LIN {X 0,Y 475.139,Z 541.907,A -85,B 0,C 180,E1 -7392.513,E2 -7392.513} C_VEL
LIN {X 0,Y 475.655,Z 532.628,A -85,B 0,C 180,E1 -7393.892,E2 -7393.892} C_VEL
LIN {X 0,Y 476.259,Z 522.288,A -85,B 0,C 180,E1 -7395.184,E2 -7395.184} C_VEL
LIN {X 0,Y 476.842,Z 512.087,A -85,B 0,C 180,E1 -7396.261,E2 -7396.261} C_VEL
LIN {X 0,Y 477.486,Z 500.079,A -85,B 0,C 180,E1 -7397.34,E2 -7397.34} C_VEL
LIN {X 0,Y 478.192,Z 487.079,A -85,B 0,C 180,E1 -7398.309,E2 -7398.309} C_VEL
LIN {X 0,Y 478.818,Z 472.829,A -85,B 0,C 180,E1 -7399.172,E2 -7399.172} C_VEL
LIN {X 0,Y 479.382,Z 458.904,A -85,B 0,C 180,E1 -7399.836,E2 -7399.836} C_VEL
LIN {X 0,Y 479.815,Z 443.461,A -85,B 0,C 180,E1 -7400.392,E2 -7400.392} C_VEL
LIN {X 0,Y 480.139,Z 428.432,A -85,B 0,C 180,E1 -7400.762,E2 -7400.762} C_VEL
LIN {X 0,Y 482.379,Z 286.852,A -85,B 0,C 180,E1 -7403.143,E2 -7403.143} C_VEL
LIN {X 0,Y 481.637,Z 283.318,A -85,B 0,C 180,E1 -7403.243,E2 -7403.243} C_VEL
LIN {X 0,Y 475.324,Z 267.213,A -85,B 0,C 180,E1 -7403.872,E2 -7403.872} C_VEL
LIN {X 0,Y 474.641,Z 263.989,A -85,B 0,C 180,E1 -7404.493,E2 -7404.493} C_VEL
LIN {X 0,Y 474.638,Z 263.985,A -85,B 0,C 180,E1 -7407.323,E2 -7407.323} C_VEL
LIN {X 0,Y 474.602,Z 263.992,A -85,B 0,C 180,E1 -7410.229,E2 -7410.229} C_VEL
LIN {X 0,Y 474.643,Z 263.982,A -85,B 0,C 180,E1 -7413.219,E2 -7413.219} C_VEL
LIN {X 0,Y 474.583,Z 263.992,A -85,B 0,C 180,E1 -7416.323,E2 -7416.323} C_VEL
LIN {X 0,Y 474.624,Z 263.988,A -85,B 0,C 180,E1 -7419.547,E2 -7419.547} C_VEL
LIN {X 0,Y 474.599,Z 263.99,A -85,B 0,C 180,E1 -7422.232,E2 -7422.232} C_VEL
LIN {X 0,Y 474.615,Z 263.987,A -85,B 0,C 180,E1 -7425.296,E2 -7425.296} C_VEL
LIN {X 0,Y 474.616,Z 263.989,A -85,B 0,C 180,E1 -7428.075,E2 -7428.075} C_VEL
LIN {X 0,Y 473.952,Z 264.07,A -85,B 0,C 180,E1 -7428.783,E2 -7428.783} C_VEL
LIN {X 0,Y 471.081,Z 264.432,A -85,B 0,C 180,E1 -7429.933,E2 -7429.933} C_VEL
LIN {X 0,Y 468.659,Z 264.731,A -85,B 0,C 180,E1 -7430.86,E2 -7430.86} C_VEL
LIN {X 0,Y 467.632,Z 264.86,A -85,B 0,C 180,E1 -7431.576,E2 -7431.576} C_VEL
LIN {X 0,Y 467.557,Z 264.869,A -85,B 0,C 180,E1 -7431.819,E2 -7431.819} C_VEL
LIN {X 0,Y 467.554,Z 264.866,A -85,B 0,C 180,E1 -7435.166,E2 -7435.166} C_VEL
LIN {X 0,Y 467.578,Z 264.864,A -85,B 0,C 180,E1 -7438.259,E2 -7438.259} C_VEL
LIN {X 0,Y 467.551,Z 264.867,A -85,B 0,C 180,E1 -7441.248,E2 -7441.248} C_VEL
LIN {X 0,Y 467.58,Z 264.864,A -85,B 0,C 180,E1 -7444.157,E2 -7444.157} C_VEL
LIN {X 0,Y 467.571,Z 264.863,A -85,B 0,C 180,E1 -7446.995,E2 -7446.995} C_VEL
LIN {X 0,Y 467.617,Z 264.864,A -85,B 0,C 180,E1 -7449.776,E2 -7449.776} C_VEL
LIN {X 0,Y 467.592,Z 264.86,A -85,B 0,C 180,E1 -7452.505,E2 -7452.505} C_VEL
LIN {X 0,Y 467.599,Z 264.862,A -85,B 0,C 180,E1 -7455.195,E2 -7455.195} C_VEL
LIN {X 0,Y 467.649,Z 264.858,A -85,B 0,C 180,E1 -7457.853,E2 -7457.853} C_VEL
LIN {X 0,Y 467.674,Z 264.855,A -85,B 0,C 180,E1 -7461.356,E2 -7461.356} C_VEL
LIN {X 0,Y 467.726,Z 264.847,A -85,B 0,C 180,E1 -7463.961,E2 -7463.961} C_VEL
LIN {X 0,Y 467.849,Z 264.834,A -85,B 0,C 180,E1 -7467.416,E2 -7467.416} C_VEL
LIN {X 0,Y 467.872,Z 264.828,A -85,B 0,C 180,E1 -7469.999,E2 -7469.999} C_VEL
LIN {X 0,Y 467.849,Z 264.828,A -85,B 0,C 180,E1 -7472.582,E2 -7472.582} C_VEL
LIN {X 0,Y 467.724,Z 264.845,A -85,B 0,C 180,E1 -7476.036,E2 -7476.036} C_VEL
LIN {X 0,Y 467.67,Z 264.85,A -85,B 0,C 180,E1 -7478.642,E2 -7478.642} C_VEL
LIN {X 0,Y 467.645,Z 264.854,A -85,B 0,C 180,E1 -7482.144,E2 -7482.144} C_VEL
LIN {X 0,Y 467.628,Z 264.861,A -85,B 0,C 180,E1 -7485.694,E2 -7485.694} C_VEL
LIN {X 0,Y 467.605,Z 264.859,A -85,B 0,C 180,E1 -7488.764,E2 -7488.764} C_VEL
LIN {X 0,Y 467.568,Z 264.869,A -85,B 0,C 180,E1 -7491.267,E2 -7491.267} C_VEL
LIN {X 0,Y 467.55,Z 264.867,A -85,B 0,C 180,E1 -7493.943,E2 -7493.943} C_VEL
LIN {X 0,Y 467.599,Z 264.86,A -85,B 0,C 180,E1 -7496.8,E2 -7496.8} C_VEL
LIN {X 0,Y 467.541,Z 264.87,A -85,B 0,C 180,E1 -7499.737,E2 -7499.737} C_VEL
LIN {X 0,Y 467.57,Z 264.864,A -85,B 0,C 180,E1 -7502.758,E2 -7502.758} C_VEL
LIN {X 0,Y 467.542,Z 264.868,A -85,B 0,C 180,E1 -7505.889,E2 -7505.889} C_VEL
LIN {X 0,Y 467.568,Z 264.869,A -85,B 0,C 180,E1 -7509.144,E2 -7509.144} C_VEL
LIN {X 0,Y 467.572,Z 264.863,A -85,B 0,C 180,E1 -7512.566,E2 -7512.566} C_VEL
LIN {X 0,Y 467.556,Z 264.87,A -85,B 0,C 180,E1 -7515.053,E2 -7515.053} C_VEL
LIN {X 0,Y 467.575,Z 264.868,A -85,B 0,C 180,E1 -7517.44,E2 -7517.44} C_VEL
LIN {X 0,Y 467.567,Z 264.866,A -85,B 0,C 180,E1 -7520.855,E2 -7520.855} C_VEL
LIN {X 0,Y 467.547,Z 264.865,A -85,B 0,C 180,E1 -7524.26,E2 -7524.26} C_VEL
LIN {X 0,Y 467.567,Z 264.87,A -85,B 0,C 180,E1 -7527.321,E2 -7527.321} C_VEL
LIN {X 0,Y 467.555,Z 264.866,A -85,B 0,C 180,E1 -7530.667,E2 -7530.667} C_VEL
LIN {X 0,Y 467.602,Z 264.867,A -85,B 0,C 180,E1 -7533.2,E2 -7533.2} C_VEL
LIN {X 0,Y 467.577,Z 264.863,A -85,B 0,C 180,E1 -7536.468,E2 -7536.468} C_VEL
LIN {X 0,Y 467.609,Z 264.859,A -85,B 0,C 180,E1 -7539.777,E2 -7539.777} C_VEL
LIN {X 0,Y 467.594,Z 264.861,A -85,B 0,C 180,E1 -7542.507,E2 -7542.507} C_VEL
LIN {X 0,Y 467.592,Z 264.867,A -85,B 0,C 180,E1 -7545.197,E2 -7545.197} C_VEL
LIN {X 0,Y 467.641,Z 264.854,A -85,B 0,C 180,E1 -7547.855,E2 -7547.855} C_VEL
LIN {X 0,Y 467.666,Z 264.855,A -85,B 0,C 180,E1 -7551.358,E2 -7551.358} C_VEL
LIN {X 0,Y 467.721,Z 264.844,A -85,B 0,C 180,E1 -7553.963,E2 -7553.963} C_VEL
LIN {X 0,Y 467.845,Z 264.832,A -85,B 0,C 180,E1 -7557.418,E2 -7557.418} C_VEL
LIN {X 0,Y 467.867,Z 264.826,A -85,B 0,C 180,E1 -7560.001,E2 -7560.001} C_VEL
LIN {X 0,Y 467.845,Z 264.831,A -85,B 0,C 180,E1 -7562.584,E2 -7562.584} C_VEL
LIN {X 0,Y 467.721,Z 264.844,A -85,B 0,C 180,E1 -7566.038,E2 -7566.038} C_VEL
LIN {X 0,Y 467.669,Z 264.854,A -85,B 0,C 180,E1 -7568.644,E2 -7568.644} C_VEL
LIN {X 0,Y 467.644,Z 264.854,A -85,B 0,C 180,E1 -7572.146,E2 -7572.146} C_VEL
LIN {X 0,Y 467.627,Z 264.856,A -85,B 0,C 180,E1 -7575.696,E2 -7575.696} C_VEL
LIN {X 0,Y 467.606,Z 264.865,A -85,B 0,C 180,E1 -7578.766,E2 -7578.766} C_VEL
LIN {X 0,Y 467.569,Z 264.866,A -85,B 0,C 180,E1 -7581.269,E2 -7581.269} C_VEL
LIN {X 0,Y 467.56,Z 264.864,A -85,B 0,C 180,E1 -7583.944,E2 -7583.944} C_VEL
LIN {X 0,Y 467.605,Z 264.866,A -85,B 0,C 180,E1 -7586.801,E2 -7586.801} C_VEL
LIN {X 0,Y 467.544,Z 264.866,A -85,B 0,C 180,E1 -7589.739,E2 -7589.739} C_VEL
LIN {X 0,Y 467.574,Z 264.87,A -85,B 0,C 180,E1 -7592.76,E2 -7592.76} C_VEL
LIN {X 0,Y 467.544,Z 264.866,A -85,B 0,C 180,E1 -7595.891,E2 -7595.891} C_VEL
LIN {X 0,Y 467.567,Z 264.867,A -85,B 0,C 180,E1 -7599.147,E2 -7599.147} C_VEL
LIN {X 0,Y 467.579,Z 264.867,A -85,B 0,C 180,E1 -7602.568,E2 -7602.568} C_VEL
LIN {X 0,Y 467.558,Z 264.868,A -85,B 0,C 180,E1 -7605.054,E2 -7605.054} C_VEL
LIN {X 0,Y 467.582,Z 264.862,A -85,B 0,C 180,E1 -7607.441,E2 -7607.441} C_VEL
LIN {X 0,Y 467.575,Z 264.869,A -85,B 0,C 180,E1 -7610.857,E2 -7610.857} C_VEL
LIN {X 0,Y 467.552,Z 264.868,A -85,B 0,C 180,E1 -7614.263,E2 -7614.263} C_VEL
LIN {X 0,Y 467.577,Z 264.864,A -85,B 0,C 180,E1 -7617.322,E2 -7617.322} C_VEL
LIN {X 0,Y 467.622,Z 265.064,A -85,B 0,C 180,E1 -7618.201,E2 -7618.201} C_VEL
LIN {X 0,Y 472.061,Z 282.686,A -85,B 0,C 180,E1 -7621.036,E2 -7621.036} C_VEL
LIN {X 0,Y 472.862,Z 286.344,A -85,B 0,C 180,E1 -7621.603,E2 -7621.603} C_VEL
LIN {X 0,Y 472.082,Z 301.582,A -85,B 0,C 180,E1 -7623.713,E2 -7623.713} C_VEL
LIN {X 0,Y 471.187,Z 317.709,A -85,B 0,C 180,E1 -7625.916,E2 -7625.916} C_VEL
LIN {X 0,Y 475.515,Z 342.088,A -85,B 0,C 180,E1 -7626.586,E2 -7626.586} C_VEL
LIN {X 0,Y 473.469,Z 470.629,A -85,B 0,C 180,E1 -7628.79,E2 -7628.79} C_VEL
LIN {X 0,Y 473.069,Z 489.021,A -85,B 0,C 180,E1 -7629.152,E2 -7629.152} C_VEL
LIN {X 0,Y 472.511,Z 504.975,A -85,B 0,C 180,E1 -7629.646,E2 -7629.646} C_VEL
LIN {X 0,Y 471.834,Z 520.281,A -85,B 0,C 180,E1 -7630.307,E2 -7630.307} C_VEL
LIN {X 0,Y 471.125,Z 533.944,A -85,B 0,C 180,E1 -7631.069,E2 -7631.069} C_VEL
LIN {X 0,Y 470.314,Z 548.109,A -85,B 0,C 180,E1 -7632.05,E2 -7632.05} C_VEL
LIN {X 0,Y 469.588,Z 561.022,A -85,B 0,C 180,E1 -7633.146,E2 -7633.146} C_VEL
LIN {X 0,Y 468.886,Z 572.867,A -85,B 0,C 180,E1 -7634.349,E2 -7634.349} C_VEL
LIN {X 0,Y 468.262,Z 583.736,A -85,B 0,C 180,E1 -7635.663,E2 -7635.663} C_VEL
LIN {X 0,Y 467.737,Z 592.926,A -85,B 0,C 180,E1 -7636.976,E2 -7636.976} C_VEL
LIN {X 0,Y 467.384,Z 601.953,A -85,B 0,C 180,E1 -7638.509,E2 -7638.509} C_VEL
LIN {X 0,Y 467.048,Z 609.45,A -85,B 0,C 180,E1 -7640.036,E2 -7640.036} C_VEL
LIN {X 0,Y 466.857,Z 616.377,A -85,B 0,C 180,E1 -7641.779,E2 -7641.779} C_VEL
LIN {X 0,Y 466.796,Z 620.542,A -85,B 0,C 180,E1 -7643.083,E2 -7643.083} C_VEL
LIN {X 0,Y 466.715,Z 624.893,A -85,B 0,C 180,E1 -7644.817,E2 -7644.817} C_VEL
LIN {X 0,Y 466.715,Z 627.937,A -85,B 0,C 180,E1 -7646.548,E2 -7646.548} C_VEL
LIN {X 0,Y 466.691,Z 629.731,A -85,B 0,C 180,E1 -7648.275,E2 -7648.275} C_VEL
LIN {X 0,Y 466.599,Z 630.303,A -85,B 0,C 180,E1 -7650.001,E2 -7650.001} C_VEL
LIN {X 0,Y 466.693,Z 629.626,A -85,B 0,C 180,E1 -7651.727,E2 -7651.727} C_VEL
LIN {X 0,Y 466.735,Z 627.727,A -85,B 0,C 180,E1 -7653.454,E2 -7653.454} C_VEL
LIN {X 0,Y 466.737,Z 624.572,A -85,B 0,C 180,E1 -7655.185,E2 -7655.185} C_VEL
LIN {X 0,Y 466.749,Z 620.092,A -85,B 0,C 180,E1 -7656.92,E2 -7656.92} C_VEL
LIN {X 0,Y 466.881,Z 614.167,A -85,B 0,C 180,E1 -7658.659,E2 -7658.659} C_VEL
LIN {X 0,Y 467.123,Z 606.626,A -85,B 0,C 180,E1 -7660.402,E2 -7660.402} C_VEL
LIN {X 0,Y 467.36,Z 598.534,A -85,B 0,C 180,E1 -7661.934,E2 -7661.934} C_VEL
LIN {X 0,Y 467.86,Z 588.796,A -85,B 0,C 180,E1 -7663.465,E2 -7663.465} C_VEL
LIN {X 0,Y 468.341,Z 578.857,A -85,B 0,C 180,E1 -7664.781,E2 -7664.781} C_VEL
LIN {X 0,Y 468.959,Z 567.176,A -85,B 0,C 180,E1 -7666.084,E2 -7666.084} C_VEL
LIN {X 0,Y 469.721,Z 554.071,A -85,B 0,C 180,E1 -7667.301,E2 -7667.301} C_VEL
LIN {X 0,Y 470.469,Z 541.328,A -85,B 0,C 180,E1 -7668.284,E2 -7668.284} C_VEL
LIN {X 0,Y 471.174,Z 526.601,A -85,B 0,C 180,E1 -7669.214,E2 -7669.214} C_VEL
LIN {X 0,Y 471.963,Z 511.256,A -85,B 0,C 180,E1 -7669.973,E2 -7669.973} C_VEL
LIN {X 0,Y 472.552,Z 496.207,A -85,B 0,C 180,E1 -7670.539,E2 -7670.539} C_VEL
LIN {X 0,Y 473.101,Z 480.803,A -85,B 0,C 180,E1 -7670.945,E2 -7670.945} C_VEL
LIN {X 0,Y 475.142,Z 376.079,A -85,B 0,C 180,E1 -7672.861,E2 -7672.861} C_VEL
LIN {X 0,Y 475.834,Z 341.657,A -85,B 0,C 180,E1 -7673.539,E2 -7673.539} C_VEL
LIN {X 0,Y 472.404,Z 320.404,A -85,B 0,C 180,E1 -7674.215,E2 -7674.215} C_VEL
LIN {X 0,Y 471.131,Z 313.647,A -85,B 0,C 180,E1 -7674.462,E2 -7674.462} C_VEL
LIN {X 0,Y 472.534,Z 292.625,A -85,B 0,C 180,E1 -7677.457,E2 -7677.457} C_VEL
LIN {X 0,Y 472.897,Z 286.289,A -85,B 0,C 180,E1 -7678.397,E2 -7678.397} C_VEL
LIN {X 0,Y 470.902,Z 276.797,A -85,B 0,C 180,E1 -7680.046,E2 -7680.046} C_VEL
LIN {X 0,Y 467.596,Z 264.869,A -85,B 0,C 180,E1 -7682.355,E2 -7682.355} C_VEL
LIN {X 0,Y 467.569,Z 264.872,A -85,B 0,C 180,E1 -7684.833,E2 -7684.833} C_VEL
LIN {X 0,Y 467.571,Z 264.868,A -85,B 0,C 180,E1 -7688.045,E2 -7688.045} C_VEL
LIN {X 0,Y 467.584,Z 264.868,A -85,B 0,C 180,E1 -7691.277,E2 -7691.277} C_VEL
LIN {X 0,Y 467.56,Z 264.869,A -85,B 0,C 180,E1 -7693.821,E2 -7693.821} C_VEL
LIN {X 0,Y 467.562,Z 264.87,A -85,B 0,C 180,E1 -7696.256,E2 -7696.256} C_VEL
LIN {X 0,Y 467.584,Z 264.867,A -85,B 0,C 180,E1 -7698.723,E2 -7698.723} C_VEL
LIN {X 0,Y 467.568,Z 264.868,A -85,B 0,C 180,E1 -7701.955,E2 -7701.955} C_VEL
LIN {X 0,Y 467.569,Z 264.869,A -85,B 0,C 180,E1 -7705.167,E2 -7705.167} C_VEL
LIN {X 0,Y 467.589,Z 264.868,A -85,B 0,C 180,E1 -7708.26,E2 -7708.26} C_VEL
LIN {X 0,Y 467.562,Z 264.87,A -85,B 0,C 180,E1 -7711.249,E2 -7711.249} C_VEL
LIN {X 0,Y 467.606,Z 264.969,A -85,B 0,C 180,E1 -7713.68,E2 -7713.68} C_VEL
LIN {X 0,Y 469.637,Z 272.657,A -85,B 0,C 180,E1 -7715.539,E2 -7715.539} C_VEL
LIN {X 0,Y 476.247,Z 287.026,A -85,B 0,C 180,E1 -7716.329,E2 -7716.329} C_VEL
LIN {X 0,Y 476.76,Z 288.495,A -85,B 0,C 180,E1 -7716.395,E2 -7716.395} C_VEL
LIN {X 0,Y 474.275,Z 384.716,A -85,B 0,C 180,E1 -7718.256,E2 -7718.256} C_VEL
LIN {X 0,Y 473.345,Z 436.186,A -85,B 0,C 180,E1 -7719.213,E2 -7719.213} C_VEL
LIN {X 0,Y 472.938,Z 451.934,A -85,B 0,C 180,E1 -7719.683,E2 -7719.683} C_VEL
LIN {X 0,Y 472.36,Z 467.317,A -85,B 0,C 180,E1 -7720.328,E2 -7720.328} C_VEL
LIN {X 0,Y 471.792,Z 481.298,A -85,B 0,C 180,E1 -7721.095,E2 -7721.095} C_VEL
LIN {X 0,Y 471.139,Z 494.235,A -85,B 0,C 180,E1 -7721.969,E2 -7721.969} C_VEL
LIN {X 0,Y 470.398,Z 506.614,A -85,B 0,C 180,E1 -7722.98,E2 -7722.98} C_VEL
LIN {X 0,Y 469.693,Z 518.511,A -85,B 0,C 180,E1 -7724.152,E2 -7724.152} C_VEL
LIN {X 0,Y 469.09,Z 529.643,A -85,B 0,C 180,E1 -7725.466,E2 -7725.466} C_VEL
LIN {X 0,Y 468.432,Z 539.004,A -85,B 0,C 180,E1 -7726.773,E2 -7726.773} C_VEL
LIN {X 0,Y 468.011,Z 548.131,A -85,B 0,C 180,E1 -7728.303,E2 -7728.303} C_VEL
LIN {X 0,Y 467.538,Z 555.678,A -85,B 0,C 180,E1 -7729.826,E2 -7729.826} C_VEL
LIN {X 0,Y 467.245,Z 561.874,A -85,B 0,C 180,E1 -7731.349,E2 -7731.349} C_VEL
LIN {X 0,Y 467.029,Z 567.516,A -85,B 0,C 180,E1 -7733.085,E2 -7733.085} C_VEL
LIN {X 0,Y 466.78,Z 571.769,A -85,B 0,C 180,E1 -7734.816,E2 -7734.816} C_VEL
LIN {X 0,Y 466.809,Z 574.726,A -85,B 0,C 180,E1 -7736.547,E2 -7736.547} C_VEL
LIN {X 0,Y 466.698,Z 576.487,A -85,B 0,C 180,E1 -7738.273,E2 -7738.273} C_VEL
LIN {X 0,Y 466.603,Z 577.058,A -85,B 0,C 180,E1 -7739.999,E2 -7739.999} C_VEL
LIN {X 0,Y 466.698,Z 576.411,A -85,B 0,C 180,E1 -7741.725,E2 -7741.725} C_VEL
LIN {X 0,Y 466.798,Z 574.598,A -85,B 0,C 180,E1 -7743.452,E2 -7743.452} C_VEL
LIN {X 0,Y 466.771,Z 571.587,A -85,B 0,C 180,E1 -7745.182,E2 -7745.182} C_VEL
LIN {X 0,Y 466.964,Z 568.154,A -85,B 0,C 180,E1 -7746.618,E2 -7746.618} C_VEL
LIN {X 0,Y 467.113,Z 563.187,A -85,B 0,C 180,E1 -7748.217,E2 -7748.217} C_VEL
LIN {X 0,Y 467.403,Z 556.372,A -85,B 0,C 180,E1 -7749.957,E2 -7749.957} C_VEL
LIN {X 0,Y 467.875,Z 547.853,A -85,B 0,C 180,E1 -7751.699,E2 -7751.699} C_VEL
LIN {X 0,Y 468.343,Z 538.722,A -85,B 0,C 180,E1 -7753.228,E2 -7753.228} C_VEL
LIN {X 0,Y 469.019,Z 527.697,A -85,B 0,C 180,E1 -7754.757,E2 -7754.757} C_VEL
LIN {X 0,Y 469.682,Z 516.311,A -85,B 0,C 180,E1 -7756.07,E2 -7756.07} C_VEL
LIN {X 0,Y 470.414,Z 504.354,A -85,B 0,C 180,E1 -7757.222,E2 -7757.222} C_VEL
LIN {X 0,Y 471.102,Z 491.472,A -85,B 0,C 180,E1 -7758.256,E2 -7758.256} C_VEL
LIN {X 0,Y 471.777,Z 478.174,A -85,B 0,C 180,E1 -7759.13,E2 -7759.13} C_VEL
LIN {X 0,Y 472.413,Z 464.765,A -85,B 0,C 180,E1 -7759.838,E2 -7759.838} C_VEL
LIN {X 0,Y 472.915,Z 449.672,A -85,B 0,C 180,E1 -7760.459,E2 -7760.459} C_VEL
LIN {X 0,Y 473.314,Z 435.541,A -85,B 0,C 180,E1 -7760.876,E2 -7760.876} C_VEL
LIN {X 0,Y 473.668,Z 413.779,A -85,B 0,C 180,E1 -7761.287,E2 -7761.287} C_VEL
LIN {X 0,Y 475.785,Z 287.085,A -85,B 0,C 180,E1 -7763.464,E2 -7763.464} C_VEL
LIN {X 0,Y 468.175,Z 267.585,A -85,B 0,C 180,E1 -7764.228,E2 -7764.228} C_VEL
LIN {X 0,Y 467.608,Z 264.865,A -85,B 0,C 180,E1 -7764.768,E2 -7764.768} C_VEL
LIN {X 0,Y 467.581,Z 264.868,A -85,B 0,C 180,E1 -7767.77,E2 -7767.77} C_VEL
LIN {X 0,Y 467.567,Z 264.865,A -85,B 0,C 180,E1 -7771.043,E2 -7771.043} C_VEL
LIN {X 0,Y 467.588,Z 264.864,A -85,B 0,C 180,E1 -7774.241,E2 -7774.241} C_VEL
LIN {X 0,Y 467.542,Z 264.867,A -85,B 0,C 180,E1 -7777.184,E2 -7777.184} C_VEL
LIN {X 0,Y 467.569,Z 264.866,A -85,B 0,C 180,E1 -7780.264,E2 -7780.264} C_VEL
LIN {X 0,Y 467.547,Z 264.873,A -85,B 0,C 180,E1 -7783.744,E2 -7783.744} C_VEL
LIN {X 0,Y 467.549,Z 264.868,A -85,B 0,C 180,E1 -7786.254,E2 -7786.254} C_VEL
LIN {X 0,Y 467.576,Z 264.862,A -85,B 0,C 180,E1 -7788.722,E2 -7788.722} C_VEL
LIN {X 0,Y 467.557,Z 264.869,A -85,B 0,C 180,E1 -7791.819,E2 -7791.819} C_VEL
LIN {X 0,Y 466.897,Z 264.955,A -85,B 0,C 180,E1 -7792.538,E2 -7792.538} C_VEL
LIN {X 0,Y 464.007,Z 265.314,A -85,B 0,C 180,E1 -7793.705,E2 -7793.705} C_VEL
LIN {X 0,Y 461.585,Z 265.61,A -85,B 0,C 180,E1 -7794.647,E2 -7794.647} C_VEL
LIN {X 0,Y 460.589,Z 265.736,A -85,B 0,C 180,E1 -7795.375,E2 -7795.375} C_VEL
LIN {X 0,Y 460.533,Z 265.746,A -85,B 0,C 180,E1 -7795.621,E2 -7795.621} C_VEL
LIN {X 0,Y 460.533,Z 265.739,A -85,B 0,C 180,E1 -7798.743,E2 -7798.743} C_VEL
LIN {X 0,Y 460.546,Z 265.739,A -85,B 0,C 180,E1 -7802.26,E2 -7802.26} C_VEL
LIN {X 0,Y 460.535,Z 265.739,A -85,B 0,C 180,E1 -7804.703,E2 -7804.703} C_VEL
LIN {X 0,Y 460.505,Z 265.749,A -85,B 0,C 180,E1 -7807.57,E2 -7807.57} C_VEL
LIN {X 0,Y 460.562,Z 265.736,A -85,B 0,C 180,E1 -7810.383,E2 -7810.383} C_VEL
LIN {X 0,Y 460.594,Z 265.735,A -85,B 0,C 180,E1 -7814.001,E2 -7814.001} C_VEL
LIN {X 0,Y 460.602,Z 265.739,A -85,B 0,C 180,E1 -7817.665,E2 -7817.665} C_VEL
LIN {X 0,Y 460.621,Z 265.732,A -85,B 0,C 180,E1 -7821.223,E2 -7821.223} C_VEL
LIN {X 0,Y 460.692,Z 265.724,A -85,B 0,C 180,E1 -7823.869,E2 -7823.869} C_VEL
LIN {X 0,Y 460.79,Z 265.713,A -85,B 0,C 180,E1 -7827.376,E2 -7827.376} C_VEL
LIN {X 0,Y 460.843,Z 265.703,A -85,B 0,C 180,E1 -7829.999,E2 -7829.999} C_VEL
LIN {X 0,Y 460.79,Z 265.707,A -85,B 0,C 180,E1 -7832.621,E2 -7832.621} C_VEL
LIN {X 0,Y 460.691,Z 265.721,A -85,B 0,C 180,E1 -7836.129,E2 -7836.129} C_VEL
LIN {X 0,Y 460.617,Z 265.729,A -85,B 0,C 180,E1 -7838.775,E2 -7838.775} C_VEL
LIN {X 0,Y 460.603,Z 265.731,A -85,B 0,C 180,E1 -7842.444,E2 -7842.444} C_VEL
LIN {X 0,Y 460.589,Z 265.734,A -85,B 0,C 180,E1 -7845.997,E2 -7845.997} C_VEL
LIN {X 0,Y 460.559,Z 265.738,A -85,B 0,C 180,E1 -7848.901,E2 -7848.901} C_VEL
LIN {X 0,Y 460.503,Z 265.751,A -85,B 0,C 180,E1 -7851.485,E2 -7851.485} C_VEL
LIN {X 0,Y 460.518,Z 265.741,A -85,B 0,C 180,E1 -7854.332,E2 -7854.332} C_VEL
LIN {X 0,Y 460.575,Z 265.737,A -85,B 0,C 180,E1 -7857.747,E2 -7857.747} C_VEL
LIN {X 0,Y 460.509,Z 265.749,A -85,B 0,C 180,E1 -7861.283,E2 -7861.283} C_VEL
LIN {X 0,Y 460.52,Z 265.741,A -85,B 0,C 180,E1 -7864.505,E2 -7864.505} C_VEL
LIN {X 0,Y 460.514,Z 265.746,A -85,B 0,C 180,E1 -7867.62,E2 -7867.62} C_VEL
LIN {X 0,Y 460.528,Z 265.74,A -85,B 0,C 180,E1 -7870.269,E2 -7870.269} C_VEL
LIN {X 0,Y 460.495,Z 265.751,A -85,B 0,C 180,E1 -7873.374,E2 -7873.374} C_VEL
LIN {X 0,Y 460.497,Z 265.745,A -85,B 0,C 180,E1 -7876.626,E2 -7876.626} C_VEL
LIN {X 0,Y 460.527,Z 265.742,A -85,B 0,C 180,E1 -7879.73,E2 -7879.73} C_VEL
LIN {X 0,Y 460.485,Z 265.746,A -85,B 0,C 180,E1 -7882.523,E2 -7882.523} C_VEL
LIN {X 0,Y 460.533,Z 265.742,A -85,B 0,C 180,E1 -7885.624,E2 -7885.624} C_VEL
LIN {X 0,Y 460.522,Z 265.743,A -85,B 0,C 180,E1 -7888.745,E2 -7888.745} C_VEL
LIN {X 0,Y 460.566,Z 265.735,A -85,B 0,C 180,E1 -7892.254,E2 -7892.254} C_VEL
LIN {X 0,Y 460.543,Z 265.74,A -85,B 0,C 180,E1 -7894.706,E2 -7894.706} C_VEL
LIN {X 0,Y 460.496,Z 265.747,A -85,B 0,C 180,E1 -7897.572,E2 -7897.572} C_VEL
LIN {X 0,Y 460.555,Z 265.737,A -85,B 0,C 180,E1 -7900.385,E2 -7900.385} C_VEL
LIN {X 0,Y 460.55,Z 265.745,A -85,B 0,C 180,E1 -7903.147,E2 -7903.147} C_VEL
LIN {X 0,Y 460.539,Z 265.739,A -85,B 0,C 180,E1 -7905.868,E2 -7905.868} C_VEL
LIN {X 0,Y 460.596,Z 265.733,A -85,B 0,C 180,E1 -7908.56,E2 -7908.56} C_VEL
LIN {X 0,Y 460.681,Z 265.721,A -85,B 0,C 180,E1 -7912.109,E2 -7912.109} C_VEL
LIN {X 0,Y 460.678,Z 265.725,A -85,B 0,C 180,E1 -7914.749,E2 -7914.749} C_VEL
LIN {X 0,Y 460.81,Z 265.708,A -85,B 0,C 180,E1 -7917.378,E2 -7917.378} C_VEL
LIN {X 0,Y 460.838,Z 265.701,A -85,B 0,C 180,E1 -7920.001,E2 -7920.001} C_VEL
LIN {X 0,Y 460.786,Z 265.711,A -85,B 0,C 180,E1 -7922.623,E2 -7922.623} C_VEL
LIN {X 0,Y 460.688,Z 265.72,A -85,B 0,C 180,E1 -7926.131,E2 -7926.131} C_VEL
LIN {X 0,Y 460.616,Z 265.734,A -85,B 0,C 180,E1 -7928.777,E2 -7928.777} C_VEL
LIN {X 0,Y 460.601,Z 265.733,A -85,B 0,C 180,E1 -7932.446,E2 -7932.446} C_VEL
LIN {X 0,Y 460.588,Z 265.732,A -85,B 0,C 180,E1 -7935.999,E2 -7935.999} C_VEL
LIN {X 0,Y 460.56,Z 265.744,A -85,B 0,C 180,E1 -7938.903,E2 -7938.903} C_VEL
LIN {X 0,Y 460.505,Z 265.744,A -85,B 0,C 180,E1 -7941.487,E2 -7941.487} C_VEL
LIN {X 0,Y 460.527,Z 265.742,A -85,B 0,C 180,E1 -7944.334,E2 -7944.334} C_VEL
LIN {X 0,Y 460.562,Z 265.739,A -85,B 0,C 180,E1 -7947.245,E2 -7947.245} C_VEL
LIN {X 0,Y 460.501,Z 265.745,A -85,B 0,C 180,E1 -7950.241,E2 -7950.241} C_VEL
LIN {X 0,Y 460.519,Z 265.743,A -85,B 0,C 180,E1 -7953.326,E2 -7953.326} C_VEL
LIN {X 0,Y 460.467,Z 265.752,A -85,B 0,C 180,E1 -7956.531,E2 -7956.531} C_VEL
LIN {X 0,Y 460.518,Z 265.741,A -85,B 0,C 180,E1 -7959.864,E2 -7959.864} C_VEL
LIN {X 0,Y 460.505,Z 265.749,A -85,B 0,C 180,E1 -7962.902,E2 -7962.902} C_VEL
LIN {X 0,Y 460.501,Z 265.743,A -85,B 0,C 180,E1 -7965.832,E2 -7965.832} C_VEL
LIN {X 0,Y 460.524,Z 265.747,A -85,B 0,C 180,E1 -7968.99,E2 -7968.99} C_VEL
LIN {X 0,Y 460.519,Z 265.745,A -85,B 0,C 180,E1 -7971.268,E2 -7971.268} C_VEL
LIN {X 0,Y 460.503,Z 265.747,A -85,B 0,C 180,E1 -7974.556,E2 -7974.556} C_VEL
LIN {X 0,Y 460.566,Z 265.837,A -85,B 0,C 180,E1 -7977.863,E2 -7977.863} C_VEL
LIN {X 0,Y 465.166,Z 284.085,A -85,B 0,C 180,E1 -7980.842,E2 -7980.842} C_VEL
LIN {X 0,Y 466.072,Z 289.256,A -85,B 0,C 180,E1 -7981.643,E2 -7981.643} C_VEL
LIN {X 0,Y 464.688,Z 312.945,A -85,B 0,C 180,E1 -7984.947,E2 -7984.947} C_VEL
LIN {X 0,Y 464.42,Z 317.387,A -85,B 0,C 180,E1 -7985.559,E2 -7985.559} C_VEL
LIN {X 0,Y 468.902,Z 342.971,A -85,B 0,C 180,E1 -7986.277,E2 -7986.277} C_VEL
LIN {X 0,Y 466.793,Z 467.854,A -85,B 0,C 180,E1 -7988.472,E2 -7988.472} C_VEL
LIN {X 0,Y 466.329,Z 488.219,A -85,B 0,C 180,E1 -7988.871,E2 -7988.871} C_VEL
LIN {X 0,Y 465.723,Z 504.376,A -85,B 0,C 180,E1 -7989.374,E2 -7989.374} C_VEL
LIN {X 0,Y 465.085,Z 518.991,A -85,B 0,C 180,E1 -7990.009,E2 -7990.009} C_VEL
LIN {X 0,Y 464.304,Z 532.848,A -85,B 0,C 180,E1 -7990.78,E2 -7990.78} C_VEL
LIN {X 0,Y 463.467,Z 547.151,A -85,B 0,C 180,E1 -7991.776,E2 -7991.776} C_VEL
LIN {X 0,Y 462.687,Z 560.161,A -85,B 0,C 180,E1 -7992.886,E2 -7992.886} C_VEL
LIN {X 0,Y 461.949,Z 572.096,A -85,B 0,C 180,E1 -7994.108,E2 -7994.108} C_VEL
LIN {X 0,Y 461.266,Z 583.034,A -85,B 0,C 180,E1 -7995.441,E2 -7995.441} C_VEL
LIN {X 0,Y 460.656,Z 593.691,A -85,B 0,C 180,E1 -7996.997,E2 -7996.997} C_VEL
LIN {X 0,Y 460.276,Z 602.535,A -85,B 0,C 180,E1 -7998.552,E2 -7998.552} C_VEL
LIN {X 0,Y 459.98,Z 608.933,A -85,B 0,C 180,E1 -7999.881,E2 -7999.881} C_VEL
LIN {X 0,Y 459.772,Z 615.901,A -85,B 0,C 180,E1 -8001.652,E2 -8001.652} C_VEL
LIN {X 0,Y 459.715,Z 620.086,A -85,B 0,C 180,E1 -8002.976,E2 -8002.976} C_VEL
LIN {X 0,Y 459.62,Z 624.463,A -85,B 0,C 180,E1 -8004.737,E2 -8004.737} C_VEL
LIN {X 0,Y 459.628,Z 627.523,A -85,B 0,C 180,E1 -8006.495,E2 -8006.495} C_VEL
LIN {X 0,Y 459.627,Z 629.328,A -85,B 0,C 180,E1 -8008.249,E2 -8008.249} C_VEL
LIN {X 0,Y 459.53,Z 629.898,A -85,B 0,C 180,E1 -8010.001,E2 -8010.001} C_VEL
LIN {X 0,Y 459.63,Z 629.216,A -85,B 0,C 180,E1 -8011.754,E2 -8011.754} C_VEL
LIN {X 0,Y 459.646,Z 627.305,A -85,B 0,C 180,E1 -8013.508,E2 -8013.508} C_VEL
LIN {X 0,Y 459.67,Z 624.135,A -85,B 0,C 180,E1 -8015.265,E2 -8015.265} C_VEL
LIN {X 0,Y 459.691,Z 619.625,A -85,B 0,C 180,E1 -8017.026,E2 -8017.026} C_VEL
LIN {X 0,Y 459.8,Z 613.67,A -85,B 0,C 180,E1 -8018.793,E2 -8018.793} C_VEL
LIN {X 0,Y 460.078,Z 606.105,A -85,B 0,C 180,E1 -8020.564,E2 -8020.564} C_VEL
LIN {X 0,Y 460.322,Z 597.852,A -85,B 0,C 180,E1 -8022.14,E2 -8022.14} C_VEL
LIN {X 0,Y 460.85,Z 588.201,A -85,B 0,C 180,E1 -8023.674,E2 -8023.674} C_VEL
LIN {X 0,Y 461.371,Z 578.233,A -85,B 0,C 180,E1 -8025.009,E2 -8025.009} C_VEL
LIN {X 0,Y 462.009,Z 567.012,A -85,B 0,C 180,E1 -8026.282,E2 -8026.282} C_VEL
LIN {X 0,Y 462.762,Z 554.7,A -85,B 0,C 180,E1 -8027.455,E2 -8027.455} C_VEL
LIN {X 0,Y 463.548,Z 542.14,A -85,B 0,C 180,E1 -8028.452,E2 -8028.452} C_VEL
LIN {X 0,Y 464.264,Z 528.702,A -85,B 0,C 180,E1 -8029.339,E2 -8029.339} C_VEL
LIN {X 0,Y 465.063,Z 514.169,A -85,B 0,C 180,E1 -8030.109,E2 -8030.109} C_VEL
LIN {X 0,Y 465.735,Z 499.213,A -85,B 0,C 180,E1 -8030.721,E2 -8030.721} C_VEL
LIN {X 0,Y 466.351,Z 483.738,A -85,B 0,C 180,E1 -8031.177,E2 -8031.177} C_VEL
LIN {X 0,Y 468.815,Z 370.332,A -85,B 0,C 180,E1 -8033.343,E2 -8033.343} C_VEL
LIN {X 0,Y 469.561,Z 343.336,A -85,B 0,C 180,E1 -8033.887,E2 -8033.887} C_VEL
LIN {X 0,Y 466.307,Z 322.533,A -85,B 0,C 180,E1 -8034.572,E2 -8034.572} C_VEL
LIN {X 0,Y 464.456,Z 312.9,A -85,B 0,C 180,E1 -8034.949,E2 -8034.949} C_VEL
LIN {X 0,Y 465.946,Z 292.874,A -85,B 0,C 180,E1 -8037.878,E2 -8037.878} C_VEL
LIN {X 0,Y 466.237,Z 288.569,A -85,B 0,C 180,E1 -8038.529,E2 -8038.529} C_VEL
LIN {X 0,Y 464.501,Z 279.9,A -85,B 0,C 180,E1 -8040.069,E2 -8040.069} C_VEL
LIN {X 0,Y 461.527,Z 269.097,A -85,B 0,C 180,E1 -8042.207,E2 -8042.207} C_VEL
LIN {X 0,Y 460.537,Z 265.749,A -85,B 0,C 180,E1 -8042.931,E2 -8042.931} C_VEL
LIN {X 0,Y 460.503,Z 265.749,A -85,B 0,C 180,E1 -8046.015,E2 -8046.015} C_VEL
LIN {X 0,Y 460.55,Z 265.745,A -85,B 0,C 180,E1 -8048.898,E2 -8048.898} C_VEL
LIN {X 0,Y 460.529,Z 265.745,A -85,B 0,C 180,E1 -8052.182,E2 -8052.182} C_VEL
LIN {X 0,Y 460.523,Z 265.746,A -85,B 0,C 180,E1 -8055.412,E2 -8055.412} C_VEL
LIN {X 0,Y 460.538,Z 265.745,A -85,B 0,C 180,E1 -8058.398,E2 -8058.398} C_VEL
LIN {X 0,Y 460.531,Z 265.745,A -85,B 0,C 180,E1 -8061.267,E2 -8061.267} C_VEL
LIN {X 0,Y 460.515,Z 265.75,A -85,B 0,C 180,E1 -8064.554,E2 -8064.554} C_VEL
LIN {X 0,Y 460.538,Z 265.744,A -85,B 0,C 180,E1 -8067.716,E2 -8067.716} C_VEL
LIN {X 0,Y 460.533,Z 265.747,A -85,B 0,C 180,E1 -8070.768,E2 -8070.768} C_VEL
LIN {X 0,Y 460.541,Z 265.828,A -85,B 0,C 180,E1 -8073.091,E2 -8073.091} C_VEL
LIN {X 0,Y 462.697,Z 273.702,A -85,B 0,C 180,E1 -8075.043,E2 -8075.043} C_VEL
LIN {X 0,Y 469.138,Z 287.071,A -85,B 0,C 180,E1 -8075.848,E2 -8075.848} C_VEL
LIN {X 0,Y 470.442,Z 290.142,A -85,B 0,C 180,E1 -8076.009,E2 -8076.009} C_VEL
LIN {X 0,Y 467.799,Z 384.926,A -85,B 0,C 180,E1 -8077.91,E2 -8077.91} C_VEL
LIN {X 0,Y 466.754,Z 437.046,A -85,B 0,C 180,E1 -8078.912,E2 -8078.912} C_VEL
LIN {X 0,Y 466.287,Z 452.529,A -85,B 0,C 180,E1 -8079.385,E2 -8079.385} C_VEL
LIN {X 0,Y 465.689,Z 467.723,A -85,B 0,C 180,E1 -8080.034,E2 -8080.034} C_VEL
LIN {X 0,Y 465.08,Z 481.69,A -85,B 0,C 180,E1 -8080.811,E2 -8080.811} C_VEL
LIN {X 0,Y 464.403,Z 494.617,A -85,B 0,C 180,E1 -8081.698,E2 -8081.698} C_VEL
LIN {X 0,Y 463.565,Z 507.524,A -85,B 0,C 180,E1 -8082.773,E2 -8082.773} C_VEL
LIN {X 0,Y 462.845,Z 518.907,A -85,B 0,C 180,E1 -8083.911,E2 -8083.911} C_VEL
LIN {X 0,Y 462.194,Z 530.042,A -85,B 0,C 180,E1 -8085.244,E2 -8085.244} C_VEL
LIN {X 0,Y 461.517,Z 539.401,A -85,B 0,C 180,E1 -8086.571,E2 -8086.571} C_VEL
LIN {X 0,Y 461.088,Z 547.314,A -85,B 0,C 180,E1 -8087.902,E2 -8087.902} C_VEL
LIN {X 0,Y 460.579,Z 555.091,A -85,B 0,C 180,E1 -8089.449,E2 -8089.449} C_VEL
LIN {X 0,Y 460.225,Z 562.3,A -85,B 0,C 180,E1 -8091.216,E2 -8091.216} C_VEL
LIN {X 0,Y 459.992,Z 567.951,A -85,B 0,C 180,E1 -8092.979,E2 -8092.979} C_VEL
LIN {X 0,Y 459.724,Z 572.203,A -85,B 0,C 180,E1 -8094.737,E2 -8094.737} C_VEL
LIN {X 0,Y 459.742,Z 575.156,A -85,B 0,C 180,E1 -8096.494,E2 -8096.494} C_VEL
LIN {X 0,Y 459.638,Z 576.908,A -85,B 0,C 180,E1 -8098.247,E2 -8098.247} C_VEL
LIN {X 0,Y 459.534,Z 577.469,A -85,B 0,C 180,E1 -8099.999,E2 -8099.999} C_VEL
LIN {X 0,Y 459.637,Z 576.803,A -85,B 0,C 180,E1 -8101.752,E2 -8101.752} C_VEL
LIN {X 0,Y 459.73,Z 574.965,A -85,B 0,C 180,E1 -8103.505,E2 -8103.505} C_VEL
LIN {X 0,Y 459.715,Z 571.922,A -85,B 0,C 180,E1 -8105.262,E2 -8105.262} C_VEL
LIN {X 0,Y 459.921,Z 567.588,A -85,B 0,C 180,E1 -8107.021,E2 -8107.021} C_VEL
LIN {X 0,Y 460.132,Z 561.866,A -85,B 0,C 180,E1 -8108.785,E2 -8108.785} C_VEL
LIN {X 0,Y 460.455,Z 554.586,A -85,B 0,C 180,E1 -8110.553,E2 -8110.553} C_VEL
LIN {X 0,Y 460.935,Z 546.759,A -85,B 0,C 180,E1 -8112.101,E2 -8112.101} C_VEL
LIN {X 0,Y 461.464,Z 537.312,A -85,B 0,C 180,E1 -8113.653,E2 -8113.653} C_VEL
LIN {X 0,Y 462.089,Z 527.675,A -85,B 0,C 180,E1 -8114.984,E2 -8114.984} C_VEL
LIN {X 0,Y 462.825,Z 516.187,A -85,B 0,C 180,E1 -8116.314,E2 -8116.314} C_VEL
LIN {X 0,Y 463.595,Z 503.398,A -85,B 0,C 180,E1 -8117.546,E2 -8117.546} C_VEL
LIN {X 0,Y 464.307,Z 491.107,A -85,B 0,C 180,E1 -8118.533,E2 -8118.533} C_VEL
LIN {X 0,Y 465.012,Z 477.659,A -85,B 0,C 180,E1 -8119.42,E2 -8119.42} C_VEL
LIN {X 0,Y 465.7,Z 462.87,A -85,B 0,C 180,E1 -8120.194,E2 -8120.194} C_VEL
LIN {X 0,Y 466.245,Z 447.639,A -85,B 0,C 180,E1 -8120.799,E2 -8120.799} C_VEL
LIN {X 0,Y 466.679,Z 432.752,A -85,B 0,C 180,E1 -8121.216,E2 -8121.216} C_VEL
LIN {X 0,Y 469.165,Z 288.586,A -85,B 0,C 180,E1 -8123.766,E2 -8123.766} C_VEL
LIN {X 0,Y 461.003,Z 267.895,A -85,B 0,C 180,E1 -8124.6,E2 -8124.6} C_VEL
LIN {X 0,Y 460.547,Z 265.744,A -85,B 0,C 180,E1 -8125.053,E2 -8125.053} C_VEL
LIN {X 0,Y 460.527,Z 265.745,A -85,B 0,C 180,E1 -8128.234,E2 -8128.234} C_VEL
LIN {X 0,Y 460.52,Z 265.744,A -85,B 0,C 180,E1 -8131.281,E2 -8131.281} C_VEL
LIN {X 0,Y 460.531,Z 265.741,A -85,B 0,C 180,E1 -8134.504,E2 -8134.504} C_VEL
LIN {X 0,Y 460.498,Z 265.749,A -85,B 0,C 180,E1 -8137.622,E2 -8137.622} C_VEL
LIN {X 0,Y 460.526,Z 265.74,A -85,B 0,C 180,E1 -8141.01,E2 -8141.01} C_VEL
LIN {X 0,Y 460.51,Z 265.742,A -85,B 0,C 180,E1 -8144.588,E2 -8144.588} C_VEL
LIN {X 0,Y 460.521,Z 265.749,A -85,B 0,C 180,E1 -8147.817,E2 -8147.817} C_VEL
LIN {X 0,Y 460.531,Z 265.74,A -85,B 0,C 180,E1 -8151.103,E2 -8151.103} C_VEL
LIN {X 0,Y 460.505,Z 265.743,A -85,B 0,C 180,E1 -8154.553,E2 -8154.553} C_VEL
LIN {X 0,Y 460.533,Z 265.746,A -85,B 0,C 180,E1 -8155.621,E2 -8155.621} C_VEL
LIN {X 0,Y 459.93,Z 265.828,A -85,B 0,C 180,E1 -8156.351,E2 -8156.351} C_VEL
LIN {X 0,Y 457.08,Z 266.183,A -85,B 0,C 180,E1 -8157.536,E2 -8157.536} C_VEL
LIN {X 0,Y 454.621,Z 266.483,A -85,B 0,C 180,E1 -8158.492,E2 -8158.492} C_VEL
LIN {X 0,Y 453.55,Z 266.611,A -85,B 0,C 180,E1 -8159.231,E2 -8159.231} C_VEL
LIN {X 0,Y 453.457,Z 266.621,A -85,B 0,C 180,E1 -8159.482,E2 -8159.482} C_VEL
LIN {X 0,Y 453.503,Z 266.617,A -85,B 0,C 180,E1 -8162.294,E2 -8162.294} C_VEL
LIN {X 0,Y 453.495,Z 266.619,A -85,B 0,C 180,E1 -8165.263,E2 -8165.263} C_VEL
LIN {X 0,Y 453.475,Z 266.619,A -85,B 0,C 180,E1 -8168.414,E2 -8168.414} C_VEL
LIN {X 0,Y 453.516,Z 266.614,A -85,B 0,C 180,E1 -8171.007,E2 -8171.007} C_VEL
LIN {X 0,Y 453.563,Z 266.613,A -85,B 0,C 180,E1 -8173.878,E2 -8173.878} C_VEL
LIN {X 0,Y 453.557,Z 266.614,A -85,B 0,C 180,E1 -8177.47,E2 -8177.47} C_VEL
LIN {X 0,Y 453.585,Z 266.607,A -85,B 0,C 180,E1 -8181.085,E2 -8181.085} C_VEL
LIN {X 0,Y 453.66,Z 266.601,A -85,B 0,C 180,E1 -8183.773,E2 -8183.773} C_VEL
LIN {X 0,Y 453.734,Z 266.591,A -85,B 0,C 180,E1 -8187.335,E2 -8187.335} C_VEL
LIN {X 0,Y 453.813,Z 266.579,A -85,B 0,C 180,E1 -8189.999,E2 -8189.999} C_VEL
LIN {X 0,Y 453.734,Z 266.586,A -85,B 0,C 180,E1 -8192.662,E2 -8192.662} C_VEL
LIN {X 0,Y 453.659,Z 266.596,A -85,B 0,C 180,E1 -8196.224,E2 -8196.224} C_VEL
LIN {X 0,Y 453.581,Z 266.607,A -85,B 0,C 180,E1 -8198.912,E2 -8198.912} C_VEL
LIN {X 0,Y 453.553,Z 266.609,A -85,B 0,C 180,E1 -8202.528,E2 -8202.528} C_VEL
LIN {X 0,Y 453.533,Z 266.612,A -85,B 0,C 180,E1 -8206.195,E2 -8206.195} C_VEL
LIN {X 0,Y 453.508,Z 266.617,A -85,B 0,C 180,E1 -8209.04,E2 -8209.04} C_VEL
LIN {X 0,Y 453.464,Z 266.623,A -85,B 0,C 180,E1 -8211.835,E2 -8211.835} C_VEL
LIN {X 0,Y 453.488,Z 266.618,A -85,B 0,C 180,E1 -8214.734,E2 -8214.734} C_VEL
LIN {X 0,Y 453.524,Z 266.614,A -85,B 0,C 180,E1 -8217.96,E2 -8217.96} C_VEL
LIN {X 0,Y 453.453,Z 266.627,A -85,B 0,C 180,E1 -8221.525,E2 -8221.525} C_VEL
LIN {X 0,Y 453.475,Z 266.62,A -85,B 0,C 180,E1 -8224.777,E2 -8224.777} C_VEL
LIN {X 0,Y 453.459,Z 266.621,A -85,B 0,C 180,E1 -8228.31,E2 -8228.31} C_VEL
LIN {X 0,Y 453.48,Z 266.619,A -85,B 0,C 180,E1 -8230.608,E2 -8230.608} C_VEL
LIN {X 0,Y 453.449,Z 266.629,A -85,B 0,C 180,E1 -8233.245,E2 -8233.245} C_VEL
LIN {X 0,Y 453.459,Z 266.623,A -85,B 0,C 180,E1 -8235.78,E2 -8235.78} C_VEL
LIN {X 0,Y 453.468,Z 266.619,A -85,B 0,C 180,E1 -8238.209,E2 -8238.209} C_VEL
LIN {X 0,Y 453.479,Z 266.62,A -85,B 0,C 180,E1 -8240.793,E2 -8240.793} C_VEL
LIN {X 0,Y 453.441,Z 266.624,A -85,B 0,C 180,E1 -8243.917,E2 -8243.917} C_VEL
LIN {X 0,Y 453.468,Z 266.627,A -85,B 0,C 180,E1 -8247.151,E2 -8247.151} C_VEL
LIN {X 0,Y 453.46,Z 266.62,A -85,B 0,C 180,E1 -8250.268,E2 -8250.268} C_VEL
LIN {X 0,Y 453.492,Z 266.623,A -85,B 0,C 180,E1 -8253.294,E2 -8253.294} C_VEL
LIN {X 0,Y 453.487,Z 266.617,A -85,B 0,C 180,E1 -8256.239,E2 -8256.239} C_VEL
LIN {X 0,Y 453.469,Z 266.627,A -85,B 0,C 180,E1 -8259.118,E2 -8259.118} C_VEL
LIN {X 0,Y 453.497,Z 266.616,A -85,B 0,C 180,E1 -8261.945,E2 -8261.945} C_VEL
LIN {X 0,Y 453.525,Z 266.615,A -85,B 0,C 180,E1 -8264.727,E2 -8264.727} C_VEL
LIN {X 0,Y 453.545,Z 266.61,A -85,B 0,C 180,E1 -8268.379,E2 -8268.379} C_VEL
LIN {X 0,Y 453.638,Z 266.598,A -85,B 0,C 180,E1 -8271.986,E2 -8271.986} C_VEL
LIN {X 0,Y 453.652,Z 266.6,A -85,B 0,C 180,E1 -8274.667,E2 -8274.667} C_VEL
LIN {X 0,Y 453.75,Z 266.588,A -85,B 0,C 180,E1 -8277.337,E2 -8277.337} C_VEL
LIN {X 0,Y 453.809,Z 266.577,A -85,B 0,C 180,E1 -8280.001,E2 -8280.001} C_VEL
LIN {X 0,Y 453.73,Z 266.59,A -85,B 0,C 180,E1 -8282.664,E2 -8282.664} C_VEL
LIN {X 0,Y 453.656,Z 266.596,A -85,B 0,C 180,E1 -8286.226,E2 -8286.226} C_VEL
LIN {X 0,Y 453.58,Z 266.613,A -85,B 0,C 180,E1 -8288.914,E2 -8288.914} C_VEL
LIN {X 0,Y 453.551,Z 266.612,A -85,B 0,C 180,E1 -8292.53,E2 -8292.53} C_VEL
LIN {X 0,Y 453.533,Z 266.612,A -85,B 0,C 180,E1 -8296.197,E2 -8296.197} C_VEL
LIN {X 0,Y 453.509,Z 266.621,A -85,B 0,C 180,E1 -8299.042,E2 -8299.042} C_VEL
LIN {X 0,Y 453.465,Z 266.62,A -85,B 0,C 180,E1 -8301.837,E2 -8301.837} C_VEL
LIN {X 0,Y 453.496,Z 266.622,A -85,B 0,C 180,E1 -8304.736,E2 -8304.736} C_VEL
LIN {X 0,Y 453.522,Z 266.613,A -85,B 0,C 180,E1 -8307.961,E2 -8307.961} C_VEL
LIN {X 0,Y 453.456,Z 266.622,A -85,B 0,C 180,E1 -8311.526,E2 -8311.526} C_VEL
LIN {X 0,Y 453.478,Z 266.626,A -85,B 0,C 180,E1 -8314.779,E2 -8314.779} C_VEL
LIN {X 0,Y 453.454,Z 266.623,A -85,B 0,C 180,E1 -8318.313,E2 -8318.313} C_VEL
LIN {X 0,Y 453.486,Z 266.623,A -85,B 0,C 180,E1 -8320.61,E2 -8320.61} C_VEL
LIN {X 0,Y 453.447,Z 266.624,A -85,B 0,C 180,E1 -8323.245,E2 -8323.245} C_VEL
LIN {X 0,Y 453.456,Z 266.621,A -85,B 0,C 180,E1 -8325.78,E2 -8325.78} C_VEL
LIN {X 0,Y 453.472,Z 266.621,A -85,B 0,C 180,E1 -8328.211,E2 -8328.211} C_VEL
LIN {X 0,Y 453.503,Z 266.623,A -85,B 0,C 180,E1 -8330.792,E2 -8330.792} C_VEL
LIN {X 0,Y 453.445,Z 266.623,A -85,B 0,C 180,E1 -8333.918,E2 -8333.918} C_VEL
LIN {X 0,Y 453.48,Z 266.62,A -85,B 0,C 180,E1 -8337.153,E2 -8337.153} C_VEL
LIN {X 0,Y 453.529,Z 266.832,A -85,B 0,C 180,E1 -8337.553,E2 -8337.553} C_VEL
LIN {X 0,Y 458.19,Z 285.213,A -85,B 0,C 180,E1 -8340.606,E2 -8340.606} C_VEL
LIN {X 0,Y 459.273,Z 290.738,A -85,B 0,C 180,E1 -8341.479,E2 -8341.479} C_VEL
LIN {X 0,Y 457.953,Z 310.746,A -85,B 0,C 180,E1 -8344.309,E2 -8344.309} C_VEL
LIN {X 0,Y 457.641,Z 317.086,A -85,B 0,C 180,E1 -8345.202,E2 -8345.202} C_VEL
LIN {X 0,Y 462.327,Z 344.493,A -85,B 0,C 180,E1 -8345.984,E2 -8345.984} C_VEL
LIN {X 0,Y 459.924,Z 474.218,A -85,B 0,C 180,E1 -8348.31,E2 -8348.31} C_VEL
LIN {X 0,Y 459.502,Z 490.68,A -85,B 0,C 180,E1 -8348.672,E2 -8348.672} C_VEL
LIN {X 0,Y 458.863,Z 506.548,A -85,B 0,C 180,E1 -8349.207,E2 -8349.207} C_VEL
LIN {X 0,Y 458.078,Z 521.987,A -85,B 0,C 180,E1 -8349.924,E2 -8349.924} C_VEL
LIN {X 0,Y 457.297,Z 535.164,A -85,B 0,C 180,E1 -8350.707,E2 -8350.707} C_VEL
LIN {X 0,Y 456.437,Z 548.976,A -85,B 0,C 180,E1 -8351.718,E2 -8351.718} C_VEL
LIN {X 0,Y 455.572,Z 562.79,A -85,B 0,C 180,E1 -8352.957,E2 -8352.957} C_VEL
LIN {X 0,Y 454.726,Z 575.201,A -85,B 0,C 180,E1 -8354.309,E2 -8354.309} C_VEL
LIN {X 0,Y 454.101,Z 585.637,A -85,B 0,C 180,E1 -8355.664,E2 -8355.664} C_VEL
LIN {X 0,Y 453.483,Z 595.796,A -85,B 0,C 180,E1 -8357.243,E2 -8357.243} C_VEL
LIN {X 0,Y 453.132,Z 604.249,A -85,B 0,C 180,E1 -8358.822,E2 -8358.822} C_VEL
LIN {X 0,Y 452.78,Z 612.102,A -85,B 0,C 180,E1 -8360.621,E2 -8360.621} C_VEL
LIN {X 0,Y 452.641,Z 618.324,A -85,B 0,C 180,E1 -8362.417,E2 -8362.417} C_VEL
LIN {X 0,Y 452.509,Z 623.076,A -85,B 0,C 180,E1 -8364.207,E2 -8364.207} C_VEL
LIN {X 0,Y 452.477,Z 625.714,A -85,B 0,C 180,E1 -8365.547,E2 -8365.547} C_VEL
LIN {X 0,Y 452.538,Z 628.162,A -85,B 0,C 180,E1 -8367.331,E2 -8367.331} C_VEL
LIN {X 0,Y 452.487,Z 629.362,A -85,B 0,C 180,E1 -8369.111,E2 -8369.111} C_VEL
LIN {X 0,Y 452.488,Z 629.3,A -85,B 0,C 180,E1 -8370.891,E2 -8370.891} C_VEL
LIN {X 0,Y 452.558,Z 627.999,A -85,B 0,C 180,E1 -8372.671,E2 -8372.671} C_VEL
LIN {X 0,Y 452.488,Z 625.451,A -85,B 0,C 180,E1 -8374.455,E2 -8374.455} C_VEL
LIN {X 0,Y 452.565,Z 621.614,A -85,B 0,C 180,E1 -8376.242,E2 -8376.242} C_VEL
LIN {X 0,Y 452.67,Z 616.377,A -85,B 0,C 180,E1 -8378.033,E2 -8378.033} C_VEL
LIN {X 0,Y 452.802,Z 609.608,A -85,B 0,C 180,E1 -8379.832,E2 -8379.832} C_VEL
LIN {X 0,Y 453.136,Z 602.309,A -85,B 0,C 180,E1 -8381.406,E2 -8381.406} C_VEL
LIN {X 0,Y 453.562,Z 593.49,A -85,B 0,C 180,E1 -8382.985,E2 -8382.985} C_VEL
LIN {X 0,Y 454.118,Z 582.862,A -85,B 0,C 180,E1 -8384.567,E2 -8384.567} C_VEL
LIN {X 0,Y 454.83,Z 570.974,A -85,B 0,C 180,E1 -8386.035,E2 -8386.035} C_VEL
LIN {X 0,Y 455.58,Z 558.979,A -85,B 0,C 180,E1 -8387.276,E2 -8387.276} C_VEL
LIN {X 0,Y 456.399,Z 545.944,A -85,B 0,C 180,E1 -8388.403,E2 -8388.403} C_VEL
LIN {X 0,Y 457.278,Z 531.688,A -85,B 0,C 180,E1 -8389.413,E2 -8389.413} C_VEL
LIN {X 0,Y 458.153,Z 516.991,A -85,B 0,C 180,E1 -8390.25,E2 -8390.25} C_VEL
LIN {X 0,Y 458.958,Z 501.369,A -85,B 0,C 180,E1 -8390.938,E2 -8390.938} C_VEL
LIN {X 0,Y 459.631,Z 485.742,A -85,B 0,C 180,E1 -8391.438,E2 -8391.438} C_VEL
LIN {X 0,Y 460.2,Z 464.226,A -85,B 0,C 180,E1 -8391.885,E2 -8391.885} C_VEL
LIN {X 0,Y 462.286,Z 378.344,A -85,B 0,C 180,E1 -8393.564,E2 -8393.564} C_VEL
LIN {X 0,Y 463.213,Z 344.075,A -85,B 0,C 180,E1 -8394.282,E2 -8394.282} C_VEL
LIN {X 0,Y 460.127,Z 323.893,A -85,B 0,C 180,E1 -8394.977,E2 -8394.977} C_VEL
LIN {X 0,Y 457.878,Z 312.204,A -85,B 0,C 180,E1 -8395.454,E2 -8395.454} C_VEL
LIN {X 0,Y 459.404,Z 293.196,A -85,B 0,C 180,E1 -8398.311,E2 -8398.311} C_VEL
LIN {X 0,Y 459.588,Z 290.518,A -85,B 0,C 180,E1 -8398.731,E2 -8398.731} C_VEL
LIN {X 0,Y 457.621,Z 281.201,A -85,B 0,C 180,E1 -8400.452,E2 -8400.452} C_VEL
LIN {X 0,Y 454.93,Z 271.304,A -85,B 0,C 180,E1 -8402.487,E2 -8402.487} C_VEL
LIN {X 0,Y 453.506,Z 266.625,A -85,B 0,C 180,E1 -8403.559,E2 -8403.559} C_VEL
LIN {X 0,Y 453.459,Z 266.627,A -85,B 0,C 180,E1 -8406.299,E2 -8406.299} C_VEL
LIN {X 0,Y 453.511,Z 266.621,A -85,B 0,C 180,E1 -8409.449,E2 -8409.449} C_VEL
LIN {X 0,Y 453.47,Z 266.626,A -85,B 0,C 180,E1 -8412.995,E2 -8412.995} C_VEL
LIN {X 0,Y 453.472,Z 266.624,A -85,B 0,C 180,E1 -8415.779,E2 -8415.779} C_VEL
LIN {X 0,Y 453.485,Z 266.623,A -85,B 0,C 180,E1 -8418.21,E2 -8418.21} C_VEL
LIN {X 0,Y 453.5,Z 266.622,A -85,B 0,C 180,E1 -8420.794,E2 -8420.794} C_VEL
LIN {X 0,Y 453.457,Z 266.626,A -85,B 0,C 180,E1 -8423.917,E2 -8423.917} C_VEL
LIN {X 0,Y 453.489,Z 266.623,A -85,B 0,C 180,E1 -8427.151,E2 -8427.151} C_VEL
LIN {X 0,Y 453.473,Z 266.627,A -85,B 0,C 180,E1 -8430.268,E2 -8430.268} C_VEL
LIN {X 0,Y 453.539,Z 266.819,A -85,B 0,C 180,E1 -8432.485,E2 -8432.485} C_VEL
LIN {X 0,Y 455.692,Z 274.475,A -85,B 0,C 180,E1 -8434.497,E2 -8434.497} C_VEL
LIN {X 0,Y 462.083,Z 287.31,A -85,B 0,C 180,E1 -8435.336,E2 -8435.336} C_VEL
LIN {X 0,Y 464.253,Z 292.598,A -85,B 0,C 180,E1 -8435.627,E2 -8435.627} C_VEL
LIN {X 0,Y 461.351,Z 385.64,A -85,B 0,C 180,E1 -8437.555,E2 -8437.555} C_VEL
LIN {X 0,Y 460.189,Z 437.649,A -85,B 0,C 180,E1 -8438.588,E2 -8438.588} C_VEL
LIN {X 0,Y 459.704,Z 452.959,A -85,B 0,C 180,E1 -8439.066,E2 -8439.066} C_VEL
LIN {X 0,Y 459.057,Z 468.289,A -85,B 0,C 180,E1 -8439.733,E2 -8439.733} C_VEL
LIN {X 0,Y 458.414,Z 482.203,A -85,B 0,C 180,E1 -8440.521,E2 -8440.521} C_VEL
LIN {X 0,Y 457.692,Z 495.097,A -85,B 0,C 180,E1 -8441.42,E2 -8441.42} C_VEL
LIN {X 0,Y 456.84,Z 507.674,A -85,B 0,C 180,E1 -8442.481,E2 -8442.481} C_VEL
LIN {X 0,Y 456.022,Z 519.367,A -85,B 0,C 180,E1 -8443.664,E2 -8443.664} C_VEL
LIN {X 0,Y 455.319,Z 530.494,A -85,B 0,C 180,E1 -8445.016,E2 -8445.016} C_VEL
LIN {X 0,Y 454.598,Z 539.855,A -85,B 0,C 180,E1 -8446.363,E2 -8446.363} C_VEL
LIN {X 0,Y 454.114,Z 547.769,A -85,B 0,C 180,E1 -8447.713,E2 -8447.713} C_VEL
LIN {X 0,Y 453.594,Z 555.544,A -85,B 0,C 180,E1 -8449.284,E2 -8449.284} C_VEL
LIN {X 0,Y 453.218,Z 562.756,A -85,B 0,C 180,E1 -8451.079,E2 -8451.079} C_VEL
LIN {X 0,Y 452.942,Z 568.405,A -85,B 0,C 180,E1 -8452.869,E2 -8452.869} C_VEL
LIN {X 0,Y 452.886,Z 570.69,A -85,B 0,C 180,E1 -8453.763,E2 -8453.763} C_VEL
LIN {X 0,Y 452.68,Z 574.278,A -85,B 0,C 180,E1 -8455.547,E2 -8455.547} C_VEL
LIN {X 0,Y 452.66,Z 576.613,A -85,B 0,C 180,E1 -8457.33,E2 -8457.33} C_VEL
LIN {X 0,Y 452.492,Z 577.765,A -85,B 0,C 180,E1 -8459.109,E2 -8459.109} C_VEL
LIN {X 0,Y 452.492,Z 577.689,A -85,B 0,C 180,E1 -8460.889,E2 -8460.889} C_VEL
LIN {X 0,Y 452.621,Z 576.41,A -85,B 0,C 180,E1 -8462.669,E2 -8462.669} C_VEL
LIN {X 0,Y 452.623,Z 573.946,A -85,B 0,C 180,E1 -8464.452,E2 -8464.452} C_VEL
LIN {X 0,Y 452.823,Z 570.222,A -85,B 0,C 180,E1 -8466.236,E2 -8466.236} C_VEL
LIN {X 0,Y 452.94,Z 565.166,A -85,B 0,C 180,E1 -8468.027,E2 -8468.027} C_VEL
LIN {X 0,Y 453.26,Z 558.632,A -85,B 0,C 180,E1 -8469.82,E2 -8469.82} C_VEL
LIN {X 0,Y 453.75,Z 550.417,A -85,B 0,C 180,E1 -8471.615,E2 -8471.615} C_VEL
LIN {X 0,Y 454.281,Z 541.475,A -85,B 0,C 180,E1 -8473.214,E2 -8473.214} C_VEL
LIN {X 0,Y 454.928,Z 531.006,A -85,B 0,C 180,E1 -8474.767,E2 -8474.767} C_VEL
LIN {X 0,Y 455.609,Z 520.08,A -85,B 0,C 180,E1 -8476.12,E2 -8476.12} C_VEL
LIN {X 0,Y 456.369,Z 508.819,A -85,B 0,C 180,E1 -8477.292,E2 -8477.292} C_VEL
LIN {X 0,Y 457.147,Z 496.515,A -85,B 0,C 180,E1 -8478.37,E2 -8478.37} C_VEL
LIN {X 0,Y 457.993,Z 482.441,A -85,B 0,C 180,E1 -8479.38,E2 -8479.38} C_VEL
LIN {X 0,Y 458.731,Z 467.741,A -85,B 0,C 180,E1 -8480.222,E2 -8480.222} C_VEL
LIN {X 0,Y 459.323,Z 452.251,A -85,B 0,C 180,E1 -8480.904,E2 -8480.904} C_VEL
LIN {X 0,Y 459.796,Z 436.661,A -85,B 0,C 180,E1 -8481.397,E2 -8481.397} C_VEL
LIN {X 0,Y 460.232,Z 415.22,A -85,B 0,C 180,E1 -8481.822,E2 -8481.822} C_VEL
LIN {X 0,Y 462.588,Z 290.293,A -85,B 0,C 180,E1 -8484.068,E2 -8484.068} C_VEL
LIN {X 0,Y 453.804,Z 268.164,A -85,B 0,C 180,E1 -8484.992,E2 -8484.992} C_VEL
LIN {X 0,Y 453.501,Z 266.622,A -85,B 0,C 180,E1 -8485.346,E2 -8485.346} C_VEL
LIN {X 0,Y 453.493,Z 266.619,A -85,B 0,C 180,E1 -8488.712,E2 -8488.712} C_VEL
LIN {X 0,Y 453.464,Z 266.628,A -85,B 0,C 180,E1 -8491.798,E2 -8491.798} C_VEL
LIN {X 0,Y 453.479,Z 266.618,A -85,B 0,C 180,E1 -8494.988,E2 -8494.988} C_VEL
LIN {X 0,Y 453.457,Z 266.623,A -85,B 0,C 180,E1 -8498.311,E2 -8498.311} C_VEL
LIN {X 0,Y 453.492,Z 266.617,A -85,B 0,C 180,E1 -8500.608,E2 -8500.608} C_VEL
LIN {X 0,Y 453.459,Z 266.624,A -85,B 0,C 180,E1 -8504.22,E2 -8504.22} C_VEL
LIN {X 0,Y 453.459,Z 266.621,A -85,B 0,C 180,E1 -8507.003,E2 -8507.003} C_VEL
LIN {X 0,Y 453.492,Z 266.62,A -85,B 0,C 180,E1 -8509.408,E2 -8509.408} C_VEL
LIN {X 0,Y 453.446,Z 266.625,A -85,B 0,C 180,E1 -8512.226,E2 -8512.226} C_VEL
LIN {X 0,Y 453.459,Z 266.622,A -85,B 0,C 180,E1 -8515.619,E2 -8515.619} C_VEL
LIN {X 0,Y 453.461,Z 266.621,A -85,B 0,C 180,E1 -8518.474,E2 -8518.474} C_VEL
LIN {X 0,Y 453.457,Z 266.621,A -85,B 0,C 180,E1 -8519.482,E2 -8519.482} C_VEL
LIN {X 0,Y 452.777,Z 266.708,A -85,B 0,C 180,E1 -8520.223,E2 -8520.223} C_VEL
LIN {X 0,Y 449.923,Z 267.065,A -85,B 0,C 180,E1 -8521.428,E2 -8521.428} C_VEL
LIN {X 0,Y 447.524,Z 267.361,A -85,B 0,C 180,E1 -8522.399,E2 -8522.399} C_VEL
LIN {X 0,Y 446.501,Z 267.489,A -85,B 0,C 180,E1 -8523.15,E2 -8523.15} C_VEL
LIN {X 0,Y 446.421,Z 267.499,A -85,B 0,C 180,E1 -8523.404,E2 -8523.404} C_VEL
LIN {X 0,Y 446.457,Z 267.498,A -85,B 0,C 180,E1 -8525.923,E2 -8525.923} C_VEL
LIN {X 0,Y 446.448,Z 267.494,A -85,B 0,C 180,E1 -8528.772,E2 -8528.772} C_VEL
LIN {X 0,Y 446.447,Z 267.502,A -85,B 0,C 180,E1 -8531.648,E2 -8531.648} C_VEL
LIN {X 0,Y 446.501,Z 267.487,A -85,B 0,C 180,E1 -8534.478,E2 -8534.478} C_VEL
LIN {X 0,Y 446.511,Z 267.488,A -85,B 0,C 180,E1 -8538.192,E2 -8538.192} C_VEL
LIN {X 0,Y 446.593,Z 267.48,A -85,B 0,C 180,E1 -8541.857,E2 -8541.857} C_VEL
LIN {X 0,Y 446.633,Z 267.471,A -85,B 0,C 180,E1 -8544.581,E2 -8544.581} C_VEL
LIN {X 0,Y 446.654,Z 267.469,A -85,B 0,C 180,E1 -8548.195,E2 -8548.195} C_VEL
LIN {X 0,Y 446.784,Z 267.455,A -85,B 0,C 180,E1 -8549.999,E2 -8549.999} C_VEL
LIN {X 0,Y 446.682,Z 267.465,A -85,B 0,C 180,E1 -8552.704,E2 -8552.704} C_VEL
LIN {X 0,Y 446.629,Z 267.472,A -85,B 0,C 180,E1 -8556.323,E2 -8556.323} C_VEL
LIN {X 0,Y 446.527,Z 267.487,A -85,B 0,C 180,E1 -8559.054,E2 -8559.054} C_VEL
LIN {X 0,Y 446.511,Z 267.487,A -85,B 0,C 180,E1 -8562.729,E2 -8562.729} C_VEL
LIN {X 0,Y 446.485,Z 267.49,A -85,B 0,C 180,E1 -8566.227,E2 -8566.227} C_VEL
LIN {X 0,Y 446.457,Z 267.499,A -85,B 0,C 180,E1 -8569.302,E2 -8569.302} C_VEL
LIN {X 0,Y 446.405,Z 267.5,A -85,B 0,C 180,E1 -8572.199,E2 -8572.199} C_VEL
LIN {X 0,Y 446.431,Z 267.501,A -85,B 0,C 180,E1 -8575.152,E2 -8575.152} C_VEL
LIN {X 0,Y 446.472,Z 267.491,A -85,B 0,C 180,E1 -8578.178,E2 -8578.178} C_VEL
LIN {X 0,Y 446.406,Z 267.502,A -85,B 0,C 180,E1 -8581.774,E2 -8581.774} C_VEL
LIN {X 0,Y 446.416,Z 267.498,A -85,B 0,C 180,E1 -8584.522,E2 -8584.522} C_VEL
LIN {X 0,Y 446.416,Z 267.498,A -85,B 0,C 180,E1 -8588.081,E2 -8588.081} C_VEL
LIN {X 0,Y 446.413,Z 267.501,A -85,B 0,C 180,E1 -8590.917,E2 -8590.917} C_VEL
LIN {X 0,Y 446.408,Z 267.501,A -85,B 0,C 180,E1 -8593.843,E2 -8593.843} C_VEL
LIN {X 0,Y 446.408,Z 267.499,A -85,B 0,C 180,E1 -8596.4,E2 -8596.4} C_VEL
LIN {X 0,Y 446.428,Z 267.498,A -85,B 0,C 180,E1 -8599.802,E2 -8599.802} C_VEL
LIN {X 0,Y 446.387,Z 267.509,A -85,B 0,C 180,E1 -8603.255,E2 -8603.255} C_VEL
LIN {X 0,Y 446.433,Z 267.497,A -85,B 0,C 180,E1 -8606.566,E2 -8606.566} C_VEL
LIN {X 0,Y 446.416,Z 267.498,A -85,B 0,C 180,E1 -8609.979,E2 -8609.979} C_VEL
LIN {X 0,Y 446.46,Z 267.496,A -85,B 0,C 180,E1 -8612.839,E2 -8612.839} C_VEL
LIN {X 0,Y 446.45,Z 267.494,A -85,B 0,C 180,E1 -8615.924,E2 -8615.924} C_VEL
LIN {X 0,Y 446.439,Z 267.498,A -85,B 0,C 180,E1 -8618.773,E2 -8618.773} C_VEL
LIN {X 0,Y 446.443,Z 267.496,A -85,B 0,C 180,E1 -8621.649,E2 -8621.649} C_VEL
LIN {X 0,Y 446.493,Z 267.489,A -85,B 0,C 180,E1 -8624.48,E2 -8624.48} C_VEL
LIN {X 0,Y 446.503,Z 267.487,A -85,B 0,C 180,E1 -8628.194,E2 -8628.194} C_VEL
LIN {X 0,Y 446.586,Z 267.477,A -85,B 0,C 180,E1 -8631.858,E2 -8631.858} C_VEL
LIN {X 0,Y 446.626,Z 267.474,A -85,B 0,C 180,E1 -8634.583,E2 -8634.583} C_VEL
LIN {X 0,Y 446.694,Z 267.468,A -85,B 0,C 180,E1 -8637.295,E2 -8637.295} C_VEL
LIN {X 0,Y 446.779,Z 267.453,A -85,B 0,C 180,E1 -8640.001,E2 -8640.001} C_VEL
LIN {X 0,Y 446.677,Z 267.469,A -85,B 0,C 180,E1 -8642.706,E2 -8642.706} C_VEL
LIN {X 0,Y 446.626,Z 267.473,A -85,B 0,C 180,E1 -8646.325,E2 -8646.325} C_VEL
LIN {X 0,Y 446.526,Z 267.491,A -85,B 0,C 180,E1 -8649.056,E2 -8649.056} C_VEL
LIN {X 0,Y 446.509,Z 267.491,A -85,B 0,C 180,E1 -8652.731,E2 -8652.731} C_VEL
LIN {X 0,Y 446.485,Z 267.49,A -85,B 0,C 180,E1 -8656.229,E2 -8656.229} C_VEL
LIN {X 0,Y 446.458,Z 267.496,A -85,B 0,C 180,E1 -8659.304,E2 -8659.304} C_VEL
LIN {X 0,Y 446.407,Z 267.5,A -85,B 0,C 180,E1 -8662.201,E2 -8662.201} C_VEL
LIN {X 0,Y 446.439,Z 267.499,A -85,B 0,C 180,E1 -8665.154,E2 -8665.154} C_VEL
LIN {X 0,Y 446.475,Z 267.491,A -85,B 0,C 180,E1 -8668.18,E2 -8668.18} C_VEL
LIN {X 0,Y 446.409,Z 267.499,A -85,B 0,C 180,E1 -8671.776,E2 -8671.776} C_VEL
LIN {X 0,Y 446.42,Z 267.502,A -85,B 0,C 180,E1 -8674.524,E2 -8674.524} C_VEL
LIN {X 0,Y 446.406,Z 267.5,A -85,B 0,C 180,E1 -8678.08,E2 -8678.08} C_VEL
LIN {X 0,Y 446.419,Z 267.504,A -85,B 0,C 180,E1 -8680.919,E2 -8680.919} C_VEL
LIN {X 0,Y 446.392,Z 267.501,A -85,B 0,C 180,E1 -8683.848,E2 -8683.848} C_VEL
LIN {X 0,Y 446.391,Z 267.505,A -85,B 0,C 180,E1 -8686.405,E2 -8686.405} C_VEL
LIN {X 0,Y 446.421,Z 267.503,A -85,B 0,C 180,E1 -8689.084,E2 -8689.084} C_VEL
LIN {X 0,Y 446.408,Z 267.501,A -85,B 0,C 180,E1 -8691.923,E2 -8691.923} C_VEL
LIN {X 0,Y 446.423,Z 267.497,A -85,B 0,C 180,E1 -8695.478,E2 -8695.478} C_VEL
LIN {X 0,Y 446.485,Z 267.637,A -85,B 0,C 180,E1 -8697.211,E2 -8697.211} C_VEL
LIN {X 0,Y 451.056,Z 285.743,A -85,B 0,C 180,E1 -8700.266,E2 -8700.266} C_VEL
LIN {X 0,Y 452.369,Z 291.551,A -85,B 0,C 180,E1 -8701.211,E2 -8701.211} C_VEL
LIN {X 0,Y 451.447,Z 306.816,A -85,B 0,C 180,E1 -8703.414,E2 -8703.414} C_VEL
LIN {X 0,Y 450.859,Z 316.849,A -85,B 0,C 180,E1 -8704.844,E2 -8704.844} C_VEL
LIN {X 0,Y 455.712,Z 345.4,A -85,B 0,C 180,E1 -8705.669,E2 -8705.669} C_VEL
LIN {X 0,Y 453.236,Z 472.436,A -85,B 0,C 180,E1 -8708.004,E2 -8708.004} C_VEL
LIN {X 0,Y 452.772,Z 489.063,A -85,B 0,C 180,E1 -8708.365,E2 -8708.365} C_VEL
LIN {X 0,Y 452.093,Z 504.651,A -85,B 0,C 180,E1 -8708.881,E2 -8708.881} C_VEL
LIN {X 0,Y 451.391,Z 519.384,A -85,B 0,C 180,E1 -8709.554,E2 -8709.554} C_VEL
LIN {X 0,Y 450.595,Z 532.105,A -85,B 0,C 180,E1 -8710.29,E2 -8710.29} C_VEL
LIN {X 0,Y 449.676,Z 546.43,A -85,B 0,C 180,E1 -8711.315,E2 -8711.315} C_VEL
LIN {X 0,Y 448.824,Z 559.47,A -85,B 0,C 180,E1 -8712.458,E2 -8712.458} C_VEL
LIN {X 0,Y 447.97,Z 571.418,A -85,B 0,C 180,E1 -8713.715,E2 -8713.715} C_VEL
LIN {X 0,Y 447.182,Z 583.21,A -85,B 0,C 180,E1 -8715.205,E2 -8715.205} C_VEL
LIN {X 0,Y 446.637,Z 592.347,A -85,B 0,C 180,E1 -8716.581,E2 -8716.581} C_VEL
LIN {X 0,Y 446.203,Z 601.321,A -85,B 0,C 180,E1 -8718.186,E2 -8718.186} C_VEL
LIN {X 0,Y 445.903,Z 607.817,A -85,B 0,C 180,E1 -8719.559,E2 -8719.559} C_VEL
LIN {X 0,Y 445.611,Z 614.879,A -85,B 0,C 180,E1 -8721.384,E2 -8721.384} C_VEL
LIN {X 0,Y 445.503,Z 620.39,A -85,B 0,C 180,E1 -8723.206,E2 -8723.206} C_VEL
LIN {X 0,Y 445.442,Z 623.552,A -85,B 0,C 180,E1 -8724.569,E2 -8724.569} C_VEL
LIN {X 0,Y 445.428,Z 626.661,A -85,B 0,C 180,E1 -8726.383,E2 -8726.383} C_VEL
LIN {X 0,Y 445.448,Z 628.5,A -85,B 0,C 180,E1 -8728.193,E2 -8728.193} C_VEL
LIN {X 0,Y 445.4,Z 629.079,A -85,B 0,C 180,E1 -8730.001,E2 -8730.001} C_VEL
LIN {X 0,Y 445.452,Z 628.394,A -85,B 0,C 180,E1 -8731.809,E2 -8731.809} C_VEL
LIN {X 0,Y 445.443,Z 626.468,A -85,B 0,C 180,E1 -8733.62,E2 -8733.62} C_VEL
LIN {X 0,Y 445.485,Z 623.277,A -85,B 0,C 180,E1 -8735.433,E2 -8735.433} C_VEL
LIN {X 0,Y 445.515,Z 618.742,A -85,B 0,C 180,E1 -8737.251,E2 -8737.251} C_VEL
LIN {X 0,Y 445.636,Z 612.741,A -85,B 0,C 180,E1 -8739.075,E2 -8739.075} C_VEL
LIN {X 0,Y 446.001,Z 605.13,A -85,B 0,C 180,E1 -8740.901,E2 -8740.901} C_VEL
LIN {X 0,Y 446.273,Z 597.146,A -85,B 0,C 180,E1 -8742.475,E2 -8742.475} C_VEL
LIN {X 0,Y 446.77,Z 588.69,A -85,B 0,C 180,E1 -8743.881,E2 -8743.881} C_VEL
LIN {X 0,Y 447.468,Z 577.143,A -85,B 0,C 180,E1 -8745.487,E2 -8745.487} C_VEL
LIN {X 0,Y 448.27,Z 565.249,A -85,B 0,C 180,E1 -8746.863,E2 -8746.863} C_VEL
LIN {X 0,Y 449.091,Z 552.242,A -85,B 0,C 180,E1 -8748.122,E2 -8748.122} C_VEL
LIN {X 0,Y 450.06,Z 539.497,A -85,B 0,C 180,E1 -8749.144,E2 -8749.144} C_VEL
LIN {X 0,Y 450.894,Z 525.804,A -85,B 0,C 180,E1 -8750.055,E2 -8750.055} C_VEL
LIN {X 0,Y 451.788,Z 510.896,A -85,B 0,C 180,E1 -8750.846,E2 -8750.846} C_VEL
LIN {X 0,Y 452.591,Z 494.782,A -85,B 0,C 180,E1 -8751.493,E2 -8751.493} C_VEL
LIN {X 0,Y 453.3,Z 478.971,A -85,B 0,C 180,E1 -8751.936,E2 -8751.936} C_VEL
LIN {X 0,Y 455.787,Z 384.348,A -85,B 0,C 180,E1 -8753.84,E2 -8753.84} C_VEL
LIN {X 0,Y 456.928,Z 344.9,A -85,B 0,C 180,E1 -8754.696,E2 -8754.696} C_VEL
LIN {X 0,Y 453.983,Z 324.975,A -85,B 0,C 180,E1 -8755.409,E2 -8755.409} C_VEL
LIN {X 0,Y 451.321,Z 311.63,A -85,B 0,C 180,E1 -8755.975,E2 -8755.975} C_VEL
LIN {X 0,Y 452.914,Z 293.627,A -85,B 0,C 180,E1 -8758.754,E2 -8758.754} C_VEL
LIN {X 0,Y 452.374,Z 289.244,A -85,B 0,C 180,E1 -8759.54,E2 -8759.54} C_VEL
LIN {X 0,Y 449.938,Z 279.169,A -85,B 0,C 180,E1 -8761.553,E2 -8761.553} C_VEL
LIN {X 0,Y 447.273,Z 270.045,A -85,B 0,C 180,E1 -8763.613,E2 -8763.613} C_VEL
LIN {X 0,Y 446.434,Z 267.505,A -85,B 0,C 180,E1 -8764.25,E2 -8764.25} C_VEL
LIN {X 0,Y 446.407,Z 267.506,A -85,B 0,C 180,E1 -8766.746,E2 -8766.746} C_VEL
LIN {X 0,Y 446.454,Z 267.499,A -85,B 0,C 180,E1 -8770.198,E2 -8770.198} C_VEL
LIN {X 0,Y 446.436,Z 267.502,A -85,B 0,C 180,E1 -8772.605,E2 -8772.605} C_VEL
LIN {X 0,Y 446.46,Z 267.499,A -85,B 0,C 180,E1 -8775.104,E2 -8775.104} C_VEL
LIN {X 0,Y 446.434,Z 267.501,A -85,B 0,C 180,E1 -8778.609,E2 -8778.609} C_VEL
LIN {X 0,Y 446.449,Z 267.5,A -85,B 0,C 180,E1 -8780.973,E2 -8780.973} C_VEL
LIN {X 0,Y 446.423,Z 267.504,A -85,B 0,C 180,E1 -8784.374,E2 -8784.374} C_VEL
LIN {X 0,Y 446.429,Z 267.502,A -85,B 0,C 180,E1 -8787.638,E2 -8787.638} C_VEL
LIN {X 0,Y 446.476,Z 267.497,A -85,B 0,C 180,E1 -8791.308,E2 -8791.308} C_VEL
LIN {X 0,Y 446.475,Z 267.572,A -85,B 0,C 180,E1 -8791.753,E2 -8791.753} C_VEL
LIN {X 0,Y 448.68,Z 275.284,A -85,B 0,C 180,E1 -8793.902,E2 -8793.902} C_VEL
LIN {X 0,Y 455.471,Z 288.39,A -85,B 0,C 180,E1 -8794.846,E2 -8794.846} C_VEL
LIN {X 0,Y 458.083,Z 294.297,A -85,B 0,C 180,E1 -8795.204,E2 -8795.204} C_VEL
LIN {X 0,Y 454.981,Z 385.473,A -85,B 0,C 180,E1 -8797.163,E2 -8797.163} C_VEL
LIN {X 0,Y 453.659,Z 438.382,A -85,B 0,C 180,E1 -8798.25,E2 -8798.25} C_VEL
LIN {X 0,Y 453.078,Z 454.225,A -85,B 0,C 180,E1 -8798.76,E2 -8798.76} C_VEL
LIN {X 0,Y 452.457,Z 469.019,A -85,B 0,C 180,E1 -8799.424,E2 -8799.424} C_VEL
LIN {X 0,Y 451.752,Z 482.845,A -85,B 0,C 180,E1 -8800.222,E2 -8800.222} C_VEL
LIN {X 0,Y 450.998,Z 495.679,A -85,B 0,C 180,E1 -8801.134,E2 -8801.134} C_VEL
LIN {X 0,Y 450.078,Z 508.403,A -85,B 0,C 180,E1 -8802.227,E2 -8802.227} C_VEL
LIN {X 0,Y 449.222,Z 519.893,A -85,B 0,C 180,E1 -8803.41,E2 -8803.41} C_VEL
LIN {X 0,Y 448.473,Z 531,A -85,B 0,C 180,E1 -8804.782,E2 -8804.782} C_VEL
LIN {X 0,Y 447.718,Z 540.359,A -85,B 0,C 180,E1 -8806.149,E2 -8806.149} C_VEL
LIN {X 0,Y 447.112,Z 549.495,A -85,B 0,C 180,E1 -8807.748,E2 -8807.748} C_VEL
LIN {X 0,Y 446.574,Z 557.038,A -85,B 0,C 180,E1 -8809.343,E2 -8809.343} C_VEL
LIN {X 0,Y 446.217,Z 563.239,A -85,B 0,C 180,E1 -8810.937,E2 -8810.937} C_VEL
LIN {X 0,Y 445.889,Z 568.88,A -85,B 0,C 180,E1 -8812.755,E2 -8812.755} C_VEL
LIN {X 0,Y 445.843,Z 571.158,A -85,B 0,C 180,E1 -8813.664,E2 -8813.664} C_VEL
LIN {X 0,Y 445.6,Z 574.738,A -85,B 0,C 180,E1 -8815.476,E2 -8815.476} C_VEL
LIN {X 0,Y 445.58,Z 577.058,A -85,B 0,C 180,E1 -8817.287,E2 -8817.287} C_VEL
LIN {X 0,Y 445.43,Z 578.188,A -85,B 0,C 180,E1 -8819.095,E2 -8819.095} C_VEL
LIN {X 0,Y 445.43,Z 578.094,A -85,B 0,C 180,E1 -8820.903,E2 -8820.903} C_VEL
LIN {X 0,Y 445.544,Z 576.786,A -85,B 0,C 180,E1 -8822.712,E2 -8822.712} C_VEL
LIN {X 0,Y 445.538,Z 574.283,A -85,B 0,C 180,E1 -8824.523,E2 -8824.523} C_VEL
LIN {X 0,Y 445.76,Z 570.515,A -85,B 0,C 180,E1 -8826.336,E2 -8826.336} C_VEL
LIN {X 0,Y 445.885,Z 565.407,A -85,B 0,C 180,E1 -8828.155,E2 -8828.155} C_VEL
LIN {X 0,Y 446.224,Z 558.811,A -85,B 0,C 180,E1 -8829.976,E2 -8829.976} C_VEL
LIN {X 0,Y 446.758,Z 550.524,A -85,B 0,C 180,E1 -8831.8,E2 -8831.8} C_VEL
LIN {X 0,Y 447.292,Z 541.626,A -85,B 0,C 180,E1 -8833.403,E2 -8833.403} C_VEL
LIN {X 0,Y 448.016,Z 530.936,A -85,B 0,C 180,E1 -8835,E2 -8835} C_VEL
LIN {X 0,Y 448.743,Z 519.899,A -85,B 0,C 180,E1 -8836.373,E2 -8836.373} C_VEL
LIN {X 0,Y 449.663,Z 507.077,A -85,B 0,C 180,E1 -8837.7,E2 -8837.7} C_VEL
LIN {X 0,Y 450.414,Z 494.598,A -85,B 0,C 180,E1 -8838.772,E2 -8838.772} C_VEL
LIN {X 0,Y 451.21,Z 481.756,A -85,B 0,C 180,E1 -8839.683,E2 -8839.683} C_VEL
LIN {X 0,Y 451.94,Z 467.903,A -85,B 0,C 180,E1 -8840.48,E2 -8840.48} C_VEL
LIN {X 0,Y 452.564,Z 452.346,A -85,B 0,C 180,E1 -8841.173,E2 -8841.173} C_VEL
LIN {X 0,Y 453.051,Z 437.497,A -85,B 0,C 180,E1 -8841.651,E2 -8841.651} C_VEL
LIN {X 0,Y 453.434,Z 418.464,A -85,B 0,C 180,E1 -8842.047,E2 -8842.047} C_VEL
LIN {X 0,Y 455.987,Z 291.934,A -85,B 0,C 180,E1 -8844.375,E2 -8844.375} C_VEL
LIN {X 0,Y 446.676,Z 268.549,A -85,B 0,C 180,E1 -8845.363,E2 -8845.363} C_VEL
LIN {X 0,Y 446.471,Z 267.497,A -85,B 0,C 180,E1 -8845.588,E2 -8845.588} C_VEL
LIN {X 0,Y 446.45,Z 267.499,A -85,B 0,C 180,E1 -8848.18,E2 -8848.18} C_VEL
LIN {X 0,Y 446.416,Z 267.501,A -85,B 0,C 180,E1 -8851.299,E2 -8851.299} C_VEL
LIN {X 0,Y 446.428,Z 267.497,A -85,B 0,C 180,E1 -8854.522,E2 -8854.522} C_VEL
LIN {X 0,Y 446.41,Z 267.504,A -85,B 0,C 180,E1 -8858.077,E2 -8858.077} C_VEL
LIN {X 0,Y 446.417,Z 267.5,A -85,B 0,C 180,E1 -8861.391,E2 -8861.391} C_VEL
LIN {X 0,Y 446.449,Z 267.494,A -85,B 0,C 180,E1 -8865.103,E2 -8865.103} C_VEL
LIN {X 0,Y 446.426,Z 267.497,A -85,B 0,C 180,E1 -8868.608,E2 -8868.608} C_VEL
LIN {X 0,Y 446.435,Z 267.496,A -85,B 0,C 180,E1 -8870.971,E2 -8870.971} C_VEL
LIN {X 0,Y 446.414,Z 267.499,A -85,B 0,C 180,E1 -8874.372,E2 -8874.372} C_VEL
LIN {X 0,Y 446.416,Z 267.504,A -85,B 0,C 180,E1 -8877.637,E2 -8877.637} C_VEL
LIN {X 0,Y 446.433,Z 267.496,A -85,B 0,C 180,E1 -8880.788,E2 -8880.788} C_VEL
LIN {X 0,Y 446.421,Z 267.499,A -85,B 0,C 180,E1 -8883.404,E2 -8883.404} C_VEL
LIN {X 0,Y 445.754,Z 267.586,A -85,B 0,C 180,E1 -8884.158,E2 -8884.158} C_VEL
LIN {X 0,Y 442.876,Z 267.943,A -85,B 0,C 180,E1 -8885.381,E2 -8885.381} C_VEL
LIN {X 0,Y 440.45,Z 268.242,A -85,B 0,C 180,E1 -8886.368,E2 -8886.368} C_VEL
LIN {X 0,Y 439.429,Z 268.37,A -85,B 0,C 180,E1 -8887.132,E2 -8887.132} C_VEL
LIN {X 0,Y 439.357,Z 268.381,A -85,B 0,C 180,E1 -8887.39,E2 -8887.39} C_VEL
LIN {X 0,Y 439.435,Z 268.367,A -85,B 0,C 180,E1 -8890.662,E2 -8890.662} C_VEL
LIN {X 0,Y 439.456,Z 268.366,A -85,B 0,C 180,E1 -8894.223,E2 -8894.223} C_VEL
LIN {X 0,Y 439.477,Z 268.366,A -85,B 0,C 180,E1 -8898,E2 -8898} C_VEL
LIN {X 0,Y 439.541,Z 268.361,A -85,B 0,C 180,E1 -8901.725,E2 -8901.725} C_VEL
LIN {X 0,Y 439.608,Z 268.346,A -85,B 0,C 180,E1 -8904.494,E2 -8904.494} C_VEL
LIN {X 0,Y 439.624,Z 268.345,A -85,B 0,C 180,E1 -8908.167,E2 -8908.167} C_VEL
LIN {X 0,Y 439.754,Z 268.33,A -85,B 0,C 180,E1 -8909.999,E2 -8909.999} C_VEL
LIN {X 0,Y 439.631,Z 268.343,A -85,B 0,C 180,E1 -8912.748,E2 -8912.748} C_VEL
LIN {X 0,Y 439.603,Z 268.347,A -85,B 0,C 180,E1 -8916.424,E2 -8916.424} C_VEL
LIN {X 0,Y 439.489,Z 268.365,A -85,B 0,C 180,E1 -8919.2,E2 -8919.2} C_VEL
LIN {X 0,Y 439.455,Z 268.367,A -85,B 0,C 180,E1 -8922.937,E2 -8922.937} C_VEL
LIN {X 0,Y 439.436,Z 268.367,A -85,B 0,C 180,E1 -8926.348,E2 -8926.348} C_VEL
LIN {X 0,Y 439.391,Z 268.378,A -85,B 0,C 180,E1 -8929.625,E2 -8929.625} C_VEL
LIN {X 0,Y 439.351,Z 268.378,A -85,B 0,C 180,E1 -8932.575,E2 -8932.575} C_VEL
LIN {X 0,Y 439.385,Z 268.379,A -85,B 0,C 180,E1 -8935.584,E2 -8935.584} C_VEL
LIN {X 0,Y 439.404,Z 268.372,A -85,B 0,C 180,E1 -8938.673,E2 -8938.673} C_VEL
LIN {X 0,Y 439.357,Z 268.378,A -85,B 0,C 180,E1 -8942.03,E2 -8942.03} C_VEL
LIN {X 0,Y 439.382,Z 268.382,A -85,B 0,C 180,E1 -8945.34,E2 -8945.34} C_VEL
LIN {X 0,Y 439.374,Z 268.376,A -85,B 0,C 180,E1 -8948.594,E2 -8948.594} C_VEL
LIN {X 0,Y 439.375,Z 268.382,A -85,B 0,C 180,E1 -8951.256,E2 -8951.256} C_VEL
LIN {X 0,Y 439.392,Z 268.375,A -85,B 0,C 180,E1 -8954.728,E2 -8954.728} C_VEL
LIN {X 0,Y 439.384,Z 268.376,A -85,B 0,C 180,E1 -8957.796,E2 -8957.796} C_VEL
LIN {X 0,Y 439.411,Z 268.371,A -85,B 0,C 180,E1 -8960.227,E2 -8960.227} C_VEL
LIN {X 0,Y 439.36,Z 268.379,A -85,B 0,C 180,E1 -8963.713,E2 -8963.713} C_VEL
LIN {X 0,Y 439.358,Z 268.383,A -85,B 0,C 180,E1 -8967.054,E2 -8967.054} C_VEL
LIN {X 0,Y 439.367,Z 268.376,A -85,B 0,C 180,E1 -8970.274,E2 -8970.274} C_VEL
LIN {X 0,Y 439.413,Z 268.375,A -85,B 0,C 180,E1 -8973.396,E2 -8973.396} C_VEL
LIN {X 0,Y 439.371,Z 268.376,A -85,B 0,C 180,E1 -8976.43,E2 -8976.43} C_VEL
LIN {X 0,Y 439.374,Z 268.38,A -85,B 0,C 180,E1 -8979.397,E2 -8979.397} C_VEL
LIN {X 0,Y 439.417,Z 268.37,A -85,B 0,C 180,E1 -8982.31,E2 -8982.31} C_VEL
LIN {X 0,Y 439.433,Z 268.375,A -85,B 0,C 180,E1 -8985.174,E2 -8985.174} C_VEL
LIN {X 0,Y 439.469,Z 268.363,A -85,B 0,C 180,E1 -8988.002,E2 -8988.002} C_VEL
LIN {X 0,Y 439.534,Z 268.356,A -85,B 0,C 180,E1 -8991.727,E2 -8991.727} C_VEL
LIN {X 0,Y 439.602,Z 268.348,A -85,B 0,C 180,E1 -8994.496,E2 -8994.496} C_VEL
LIN {X 0,Y 439.623,Z 268.344,A -85,B 0,C 180,E1 -8998.169,E2 -8998.169} C_VEL
LIN {X 0,Y 439.749,Z 268.328,A -85,B 0,C 180,E1 -9000.001,E2 -9000.001} C_VEL
LIN {X 0,Y 439.627,Z 268.348,A -85,B 0,C 180,E1 -9002.75,E2 -9002.75} C_VEL
LIN {X 0,Y 439.6,Z 268.349,A -85,B 0,C 180,E1 -9006.426,E2 -9006.426} C_VEL
LIN {X 0,Y 439.488,Z 268.366,A -85,B 0,C 180,E1 -9009.203,E2 -9009.203} C_VEL
LIN {X 0,Y 439.454,Z 268.373,A -85,B 0,C 180,E1 -9012.939,E2 -9012.939} C_VEL
LIN {X 0,Y 439.436,Z 268.369,A -85,B 0,C 180,E1 -9016.35,E2 -9016.35} C_VEL
LIN {X 0,Y 439.392,Z 268.374,A -85,B 0,C 180,E1 -9019.627,E2 -9019.627} C_VEL
LIN {X 0,Y 439.354,Z 268.382,A -85,B 0,C 180,E1 -9022.577,E2 -9022.577} C_VEL
LIN {X 0,Y 439.39,Z 268.374,A -85,B 0,C 180,E1 -9025.586,E2 -9025.586} C_VEL
LIN {X 0,Y 439.407,Z 268.377,A -85,B 0,C 180,E1 -9028.675,E2 -9028.675} C_VEL
LIN {X 0,Y 439.36,Z 268.377,A -85,B 0,C 180,E1 -9032.032,E2 -9032.032} C_VEL
LIN {X 0,Y 439.385,Z 268.375,A -85,B 0,C 180,E1 -9035.342,E2 -9035.342} C_VEL
LIN {X 0,Y 439.368,Z 268.381,A -85,B 0,C 180,E1 -9038.597,E2 -9038.597} C_VEL
LIN {X 0,Y 439.38,Z 268.376,A -85,B 0,C 180,E1 -9041.258,E2 -9041.258} C_VEL
LIN {X 0,Y 439.392,Z 268.381,A -85,B 0,C 180,E1 -9044.731,E2 -9044.731} C_VEL
LIN {X 0,Y 439.389,Z 268.373,A -85,B 0,C 180,E1 -9047.797,E2 -9047.797} C_VEL
LIN {X 0,Y 439.423,Z 268.373,A -85,B 0,C 180,E1 -9050.229,E2 -9050.229} C_VEL
LIN {X 0,Y 439.366,Z 268.377,A -85,B 0,C 180,E1 -9053.714,E2 -9053.714} C_VEL
LIN {X 0,Y 439.425,Z 268.497,A -85,B 0,C 180,E1 -9056.867,E2 -9056.867} C_VEL
LIN {X 0,Y 444.148,Z 287.097,A -85,B 0,C 180,E1 -9060.062,E2 -9060.062} C_VEL
LIN {X 0,Y 445.594,Z 294.366,A -85,B 0,C 180,E1 -9061.248,E2 -9061.248} C_VEL
LIN {X 0,Y 444.1,Z 316.857,A -85,B 0,C 180,E1 -9064.483,E2 -9064.483} C_VEL
LIN {X 0,Y 449.12,Z 346.2,A -85,B 0,C 180,E1 -9065.352,E2 -9065.352} C_VEL
LIN {X 0,Y 446.159,Z 484.378,A -85,B 0,C 180,E1 -9067.971,E2 -9067.971} C_VEL
LIN {X 0,Y 445.513,Z 500.215,A -85,B 0,C 180,E1 -9068.455,E2 -9068.455} C_VEL
LIN {X 0,Y 444.768,Z 515.497,A -85,B 0,C 180,E1 -9069.115,E2 -9069.115} C_VEL
LIN {X 0,Y 443.914,Z 528.94,A -85,B 0,C 180,E1 -9069.86,E2 -9069.86} C_VEL
LIN {X 0,Y 443.105,Z 542.341,A -85,B 0,C 180,E1 -9070.787,E2 -9070.787} C_VEL
LIN {X 0,Y 442.084,Z 556.009,A -85,B 0,C 180,E1 -9071.942,E2 -9071.942} C_VEL
LIN {X 0,Y 441.221,Z 568.338,A -85,B 0,C 180,E1 -9073.204,E2 -9073.204} C_VEL
LIN {X 0,Y 440.441,Z 579.006,A -85,B 0,C 180,E1 -9074.499,E2 -9074.499} C_VEL
LIN {X 0,Y 439.737,Z 590.219,A -85,B 0,C 180,E1 -9076.131,E2 -9076.131} C_VEL
LIN {X 0,Y 439.138,Z 598.808,A -85,B 0,C 180,E1 -9077.627,E2 -9077.627} C_VEL
LIN {X 0,Y 438.861,Z 607.209,A -85,B 0,C 180,E1 -9079.389,E2 -9079.389} C_VEL
LIN {X 0,Y 438.523,Z 614.331,A -85,B 0,C 180,E1 -9081.244,E2 -9081.244} C_VEL
LIN {X 0,Y 438.435,Z 619.886,A -85,B 0,C 180,E1 -9083.096,E2 -9083.096} C_VEL
LIN {X 0,Y 438.361,Z 623.081,A -85,B 0,C 180,E1 -9084.481,E2 -9084.481} C_VEL
LIN {X 0,Y 438.331,Z 626.218,A -85,B 0,C 180,E1 -9086.324,E2 -9086.324} C_VEL
LIN {X 0,Y 438.364,Z 628.079,A -85,B 0,C 180,E1 -9088.164,E2 -9088.164} C_VEL
LIN {X 0,Y 438.337,Z 628.663,A -85,B 0,C 180,E1 -9090.001,E2 -9090.001} C_VEL
LIN {X 0,Y 438.368,Z 627.985,A -85,B 0,C 180,E1 -9091.839,E2 -9091.839} C_VEL
LIN {X 0,Y 438.344,Z 626.062,A -85,B 0,C 180,E1 -9093.678,E2 -9093.678} C_VEL
LIN {X 0,Y 438.398,Z 622.864,A -85,B 0,C 180,E1 -9095.521,E2 -9095.521} C_VEL
LIN {X 0,Y 438.435,Z 618.32,A -85,B 0,C 180,E1 -9097.369,E2 -9097.369} C_VEL
LIN {X 0,Y 438.571,Z 612.314,A -85,B 0,C 180,E1 -9099.222,E2 -9099.222} C_VEL
LIN {X 0,Y 438.951,Z 604.682,A -85,B 0,C 180,E1 -9101.078,E2 -9101.078} C_VEL
LIN {X 0,Y 439.295,Z 596.281,A -85,B 0,C 180,E1 -9102.751,E2 -9102.751} C_VEL
LIN {X 0,Y 439.864,Z 586.676,A -85,B 0,C 180,E1 -9104.34,E2 -9104.34} C_VEL
LIN {X 0,Y 440.549,Z 576.682,A -85,B 0,C 180,E1 -9105.737,E2 -9105.737} C_VEL
LIN {X 0,Y 441.308,Z 565.82,A -85,B 0,C 180,E1 -9107.026,E2 -9107.026} C_VEL
LIN {X 0,Y 442.194,Z 553.126,A -85,B 0,C 180,E1 -9108.295,E2 -9108.295} C_VEL
LIN {X 0,Y 443.283,Z 539.107,A -85,B 0,C 180,E1 -9109.449,E2 -9109.449} C_VEL
LIN {X 0,Y 444.189,Z 525.477,A -85,B 0,C 180,E1 -9110.371,E2 -9110.371} C_VEL
LIN {X 0,Y 445.18,Z 510.221,A -85,B 0,C 180,E1 -9111.194,E2 -9111.194} C_VEL
LIN {X 0,Y 446.04,Z 494.017,A -85,B 0,C 180,E1 -9111.855,E2 -9111.855} C_VEL
LIN {X 0,Y 446.808,Z 478.342,A -85,B 0,C 180,E1 -9112.302,E2 -9112.302} C_VEL
LIN {X 0,Y 449.495,Z 384.733,A -85,B 0,C 180,E1 -9114.253,E2 -9114.253} C_VEL
LIN {X 0,Y 450.802,Z 346.384,A -85,B 0,C 180,E1 -9115.108,E2 -9115.108} C_VEL
LIN {X 0,Y 448.251,Z 328.318,A -85,B 0,C 180,E1 -9115.777,E2 -9115.777} C_VEL
LIN {X 0,Y 445.033,Z 312.276,A -85,B 0,C 180,E1 -9116.488,E2 -9116.488} C_VEL
LIN {X 0,Y 444.799,Z 310.758,A -85,B 0,C 180,E1 -9116.575,E2 -9116.575} C_VEL
LIN {X 0,Y 446.316,Z 295.696,A -85,B 0,C 180,E1 -9118.962,E2 -9118.962} C_VEL
LIN {X 0,Y 445.396,Z 289.659,A -85,B 0,C 180,E1 -9120.097,E2 -9120.097} C_VEL
LIN {X 0,Y 442.749,Z 279.182,A -85,B 0,C 180,E1 -9122.324,E2 -9122.324} C_VEL
LIN {X 0,Y 440.31,Z 271.309,A -85,B 0,C 180,E1 -9124.239,E2 -9124.239} C_VEL
LIN {X 0,Y 439.412,Z 268.38,A -85,B 0,C 180,E1 -9125.016,E2 -9125.016} C_VEL
LIN {X 0,Y 439.384,Z 268.38,A -85,B 0,C 180,E1 -9128.596,E2 -9128.596} C_VEL
LIN {X 0,Y 439.395,Z 268.379,A -85,B 0,C 180,E1 -9131.257,E2 -9131.257} C_VEL
LIN {X 0,Y 439.408,Z 268.378,A -85,B 0,C 180,E1 -9134.73,E2 -9134.73} C_VEL
LIN {X 0,Y 439.402,Z 268.376,A -85,B 0,C 180,E1 -9137.796,E2 -9137.796} C_VEL
LIN {X 0,Y 439.433,Z 268.373,A -85,B 0,C 180,E1 -9140.228,E2 -9140.228} C_VEL
LIN {X 0,Y 439.378,Z 268.38,A -85,B 0,C 180,E1 -9143.713,E2 -9143.713} C_VEL
LIN {X 0,Y 439.379,Z 268.382,A -85,B 0,C 180,E1 -9147.054,E2 -9147.054} C_VEL
LIN {X 0,Y 439.414,Z 268.378,A -85,B 0,C 180,E1 -9150.802,E2 -9150.802} C_VEL
LIN {X 0,Y 439.437,Z 268.556,A -85,B 0,C 180,E1 -9151.001,E2 -9151.001} C_VEL
LIN {X 0,Y 441.646,Z 276.182,A -85,B 0,C 180,E1 -9153.262,E2 -9153.262} C_VEL
LIN {X 0,Y 447.643,Z 287.175,A -85,B 0,C 180,E1 -9154.144,E2 -9154.144} C_VEL
LIN {X 0,Y 452.027,Z 296.606,A -85,B 0,C 180,E1 -9154.78,E2 -9154.78} C_VEL
LIN {X 0,Y 448.652,Z 385.852,A -85,B 0,C 180,E1 -9156.761,E2 -9156.761} C_VEL
LIN {X 0,Y 447.181,Z 439.313,A -85,B 0,C 180,E1 -9157.899,E2 -9157.899} C_VEL
LIN {X 0,Y 446.55,Z 455.022,A -85,B 0,C 180,E1 -9158.42,E2 -9158.42} C_VEL
LIN {X 0,Y 445.875,Z 469.922,A -85,B 0,C 180,E1 -9159.107,E2 -9159.107} C_VEL
LIN {X 0,Y 445.139,Z 483.618,A -85,B 0,C 180,E1 -9159.916,E2 -9159.916} C_VEL
LIN {X 0,Y 444.24,Z 497.773,A -85,B 0,C 180,E1 -9160.955,E2 -9160.955} C_VEL
LIN {X 0,Y 443.184,Z 510.989,A -85,B 0,C 180,E1 -9162.14,E2 -9162.14} C_VEL
LIN {X 0,Y 442.281,Z 522.435,A -85,B 0,C 180,E1 -9163.379,E2 -9163.379} C_VEL
LIN {X 0,Y 441.513,Z 533.193,A -85,B 0,C 180,E1 -9164.772,E2 -9164.772} C_VEL
LIN {X 0,Y 440.714,Z 542.31,A -85,B 0,C 180,E1 -9166.16,E2 -9166.16} C_VEL
LIN {X 0,Y 440.091,Z 551.185,A -85,B 0,C 180,E1 -9167.784,E2 -9167.784} C_VEL
LIN {X 0,Y 439.527,Z 558.555,A -85,B 0,C 180,E1 -9169.403,E2 -9169.403} C_VEL
LIN {X 0,Y 439.081,Z 565.332,A -85,B 0,C 180,E1 -9171.253,E2 -9171.253} C_VEL
LIN {X 0,Y 438.868,Z 569.374,A -85,B 0,C 180,E1 -9172.639,E2 -9172.639} C_VEL
LIN {X 0,Y 438.801,Z 571.648,A -85,B 0,C 180,E1 -9173.562,E2 -9173.562} C_VEL
LIN {X 0,Y 438.524,Z 575.213,A -85,B 0,C 180,E1 -9175.403,E2 -9175.403} C_VEL
LIN {X 0,Y 438.503,Z 577.51,A -85,B 0,C 180,E1 -9177.243,E2 -9177.243} C_VEL
LIN {X 0,Y 438.37,Z 578.613,A -85,B 0,C 180,E1 -9179.081,E2 -9179.081} C_VEL
LIN {X 0,Y 438.37,Z 578.499,A -85,B 0,C 180,E1 -9180.918,E2 -9180.918} C_VEL
LIN {X 0,Y 438.47,Z 577.156,A -85,B 0,C 180,E1 -9182.755,E2 -9182.755} C_VEL
LIN {X 0,Y 438.457,Z 574.612,A -85,B 0,C 180,E1 -9184.596,E2 -9184.596} C_VEL
LIN {X 0,Y 438.685,Z 570.794,A -85,B 0,C 180,E1 -9186.438,E2 -9186.438} C_VEL
LIN {X 0,Y 438.846,Z 565.627,A -85,B 0,C 180,E1 -9188.286,E2 -9188.286} C_VEL
LIN {X 0,Y 439.2,Z 558.964,A -85,B 0,C 180,E1 -9190.137,E2 -9190.137} C_VEL
LIN {X 0,Y 439.683,Z 551.748,A -85,B 0,C 180,E1 -9191.758,E2 -9191.758} C_VEL
LIN {X 0,Y 440.219,Z 543.306,A -85,B 0,C 180,E1 -9193.337,E2 -9193.337} C_VEL
LIN {X 0,Y 440.851,Z 534.161,A -85,B 0,C 180,E1 -9194.777,E2 -9194.777} C_VEL
LIN {X 0,Y 441.602,Z 523.664,A -85,B 0,C 180,E1 -9196.17,E2 -9196.17} C_VEL
LIN {X 0,Y 442.489,Z 511.051,A -85,B 0,C 180,E1 -9197.563,E2 -9197.563} C_VEL
LIN {X 0,Y 443.338,Z 498.409,A -85,B 0,C 180,E1 -9198.723,E2 -9198.723} C_VEL
LIN {X 0,Y 444.259,Z 484.582,A -85,B 0,C 180,E1 -9199.763,E2 -9199.763} C_VEL
LIN {X 0,Y 445.081,Z 470.268,A -85,B 0,C 180,E1 -9200.629,E2 -9200.629} C_VEL
LIN {X 0,Y 445.712,Z 454.772,A -85,B 0,C 180,E1 -9201.357,E2 -9201.357} C_VEL
LIN {X 0,Y 446.263,Z 440.119,A -85,B 0,C 180,E1 -9201.862,E2 -9201.862} C_VEL
LIN {X 0,Y 446.629,Z 423.215,A -85,B 0,C 180,E1 -9202.248,E2 -9202.248} C_VEL
LIN {X 0,Y 449.403,Z 293.615,A -85,B 0,C 180,E1 -9204.687,E2 -9204.687} C_VEL
LIN {X 0,Y 439.509,Z 268.95,A -85,B 0,C 180,E1 -9205.743,E2 -9205.743} C_VEL
LIN {X 0,Y 439.423,Z 268.374,A -85,B 0,C 180,E1 -9205.901,E2 -9205.901} C_VEL
LIN {X 0,Y 439.401,Z 268.375,A -85,B 0,C 180,E1 -9208.674,E2 -9208.674} C_VEL
LIN {X 0,Y 439.371,Z 268.383,A -85,B 0,C 180,E1 -9212.029,E2 -9212.029} C_VEL
LIN {X 0,Y 439.393,Z 268.374,A -85,B 0,C 180,E1 -9215.339,E2 -9215.339} C_VEL
LIN {X 0,Y 439.362,Z 268.377,A -85,B 0,C 180,E1 -9218.596,E2 -9218.596} C_VEL
LIN {X 0,Y 439.38,Z 268.376,A -85,B 0,C 180,E1 -9221.254,E2 -9221.254} C_VEL
LIN {X 0,Y 439.397,Z 268.372,A -85,B 0,C 180,E1 -9224.728,E2 -9224.728} C_VEL
LIN {X 0,Y 439.393,Z 268.381,A -85,B 0,C 180,E1 -9227.794,E2 -9227.794} C_VEL
LIN {X 0,Y 439.392,Z 268.376,A -85,B 0,C 180,E1 -9230.223,E2 -9230.223} C_VEL
LIN {X 0,Y 439.37,Z 268.383,A -85,B 0,C 180,E1 -9233.711,E2 -9233.711} C_VEL
LIN {X 0,Y 439.368,Z 268.377,A -85,B 0,C 180,E1 -9237.053,E2 -9237.053} C_VEL
LIN {X 0,Y 439.372,Z 268.377,A -85,B 0,C 180,E1 -9240.272,E2 -9240.272} C_VEL
LIN {X 0,Y 439.378,Z 268.379,A -85,B 0,C 180,E1 -9243.405,E2 -9243.405} C_VEL
LIN {X 0,Y 439.378,Z 268.375,A -85,B 0,C 180,E1 -9246.428,E2 -9246.428} C_VEL
LIN {X 0,Y 439.357,Z 268.381,A -85,B 0,C 180,E1 -9247.39,E2 -9247.39} C_VEL
LIN {X 0,Y 438.725,Z 268.466,A -85,B 0,C 180,E1 -9248.155,E2 -9248.155} C_VEL
LIN {X 0,Y 435.902,Z 268.816,A -85,B 0,C 180,E1 -9249.4,E2 -9249.4} C_VEL
LIN {X 0,Y 433.489,Z 269.111,A -85,B 0,C 180,E1 -9250.404,E2 -9250.404} C_VEL
LIN {X 0,Y 432.443,Z 269.241,A -85,B 0,C 180,E1 -9251.179,E2 -9251.179} C_VEL
LIN {X 0,Y 432.353,Z 269.25,A -85,B 0,C 180,E1 -9251.442,E2 -9251.442} C_VEL
LIN {X 0,Y 432.424,Z 269.245,A -85,B 0,C 180,E1 -9253.96,E2 -9253.96} C_VEL
LIN {X 0,Y 432.452,Z 269.243,A -85,B 0,C 180,E1 -9257.802,E2 -9257.802} C_VEL
LIN {X 0,Y 432.485,Z 269.241,A -85,B 0,C 180,E1 -9261.589,E2 -9261.589} C_VEL
LIN {X 0,Y 432.585,Z 269.221,A -85,B 0,C 180,E1 -9264.405,E2 -9264.405} C_VEL
LIN {X 0,Y 432.594,Z 269.221,A -85,B 0,C 180,E1 -9268.137,E2 -9268.137} C_VEL
LIN {X 0,Y 432.724,Z 269.206,A -85,B 0,C 180,E1 -9269.999,E2 -9269.999} C_VEL
LIN {X 0,Y 432.583,Z 269.222,A -85,B 0,C 180,E1 -9272.792,E2 -9272.792} C_VEL
LIN {X 0,Y 432.559,Z 269.224,A -85,B 0,C 180,E1 -9276.529,E2 -9276.529} C_VEL
LIN {X 0,Y 432.432,Z 269.246,A -85,B 0,C 180,E1 -9279.352,E2 -9279.352} C_VEL
LIN {X 0,Y 432.42,Z 269.242,A -85,B 0,C 180,E1 -9282.802,E2 -9282.802} C_VEL
LIN {X 0,Y 432.401,Z 269.244,A -85,B 0,C 180,E1 -9286.478,E2 -9286.478} C_VEL
LIN {X 0,Y 432.326,Z 269.255,A -85,B 0,C 180,E1 -9289.959,E2 -9289.959} C_VEL
LIN {X 0,Y 432.305,Z 269.258,A -85,B 0,C 180,E1 -9292.963,E2 -9292.963} C_VEL
LIN {X 0,Y 432.348,Z 269.251,A -85,B 0,C 180,E1 -9296.032,E2 -9296.032} C_VEL
LIN {X 0,Y 432.33,Z 269.258,A -85,B 0,C 180,E1 -9299.187,E2 -9299.187} C_VEL
LIN {X 0,Y 432.31,Z 269.255,A -85,B 0,C 180,E1 -9302.442,E2 -9302.442} C_VEL
LIN {X 0,Y 432.331,Z 269.257,A -85,B 0,C 180,E1 -9305.631,E2 -9305.631} C_VEL
LIN {X 0,Y 432.337,Z 269.253,A -85,B 0,C 180,E1 -9308.716,E2 -9308.716} C_VEL
LIN {X 0,Y 432.32,Z 269.256,A -85,B 0,C 180,E1 -9311.796,E2 -9311.796} C_VEL
LIN {X 0,Y 432.326,Z 269.253,A -85,B 0,C 180,E1 -9314.346,E2 -9314.346} C_VEL
LIN {X 0,Y 432.311,Z 269.259,A -85,B 0,C 180,E1 -9317.015,E2 -9317.015} C_VEL
LIN {X 0,Y 432.318,Z 269.256,A -85,B 0,C 180,E1 -9319.82,E2 -9319.82} C_VEL
LIN {X 0,Y 432.292,Z 269.262,A -85,B 0,C 180,E1 -9323.022,E2 -9323.022} C_VEL
LIN {X 0,Y 432.344,Z 269.251,A -85,B 0,C 180,E1 -9325.996,E2 -9325.996} C_VEL
LIN {X 0,Y 432.332,Z 269.256,A -85,B 0,C 180,E1 -9329.49,E2 -9329.49} C_VEL
LIN {X 0,Y 432.376,Z 269.251,A -85,B 0,C 180,E1 -9332.928,E2 -9332.928} C_VEL
LIN {X 0,Y 432.356,Z 269.25,A -85,B 0,C 180,E1 -9336.024,E2 -9336.024} C_VEL
LIN {X 0,Y 432.336,Z 269.258,A -85,B 0,C 180,E1 -9339.046,E2 -9339.046} C_VEL
LIN {X 0,Y 432.363,Z 269.249,A -85,B 0,C 180,E1 -9342.011,E2 -9342.011} C_VEL
LIN {X 0,Y 432.381,Z 269.252,A -85,B 0,C 180,E1 -9344.927,E2 -9344.927} C_VEL
LIN {X 0,Y 432.445,Z 269.239,A -85,B 0,C 180,E1 -9347.804,E2 -9347.804} C_VEL
LIN {X 0,Y 432.478,Z 269.236,A -85,B 0,C 180,E1 -9351.591,E2 -9351.591} C_VEL
LIN {X 0,Y 432.579,Z 269.223,A -85,B 0,C 180,E1 -9354.407,E2 -9354.407} C_VEL
LIN {X 0,Y 432.593,Z 269.22,A -85,B 0,C 180,E1 -9358.139,E2 -9358.139} C_VEL
LIN {X 0,Y 432.719,Z 269.204,A -85,B 0,C 180,E1 -9360.001,E2 -9360.001} C_VEL
LIN {X 0,Y 432.579,Z 269.227,A -85,B 0,C 180,E1 -9362.794,E2 -9362.794} C_VEL
LIN {X 0,Y 432.556,Z 269.227,A -85,B 0,C 180,E1 -9366.531,E2 -9366.531} C_VEL
LIN {X 0,Y 432.431,Z 269.243,A -85,B 0,C 180,E1 -9369.354,E2 -9369.354} C_VEL
LIN {X 0,Y 432.419,Z 269.248,A -85,B 0,C 180,E1 -9372.804,E2 -9372.804} C_VEL
LIN {X 0,Y 432.401,Z 269.246,A -85,B 0,C 180,E1 -9376.48,E2 -9376.48} C_VEL
LIN {X 0,Y 432.328,Z 269.253,A -85,B 0,C 180,E1 -9379.962,E2 -9379.962} C_VEL
LIN {X 0,Y 432.308,Z 269.262,A -85,B 0,C 180,E1 -9382.965,E2 -9382.965} C_VEL
LIN {X 0,Y 432.352,Z 269.25,A -85,B 0,C 180,E1 -9386.034,E2 -9386.034} C_VEL
LIN {X 0,Y 432.333,Z 269.256,A -85,B 0,C 180,E1 -9389.189,E2 -9389.189} C_VEL
LIN {X 0,Y 432.314,Z 269.258,A -85,B 0,C 180,E1 -9392.444,E2 -9392.444} C_VEL
LIN {X 0,Y 432.335,Z 269.252,A -85,B 0,C 180,E1 -9395.633,E2 -9395.633} C_VEL
LIN {X 0,Y 432.331,Z 269.259,A -85,B 0,C 180,E1 -9398.716,E2 -9398.716} C_VEL
LIN {X 0,Y 432.325,Z 269.253,A -85,B 0,C 180,E1 -9401.799,E2 -9401.799} C_VEL
LIN {X 0,Y 432.326,Z 269.256,A -85,B 0,C 180,E1 -9404.349,E2 -9404.349} C_VEL
LIN {X 0,Y 432.313,Z 269.259,A -85,B 0,C 180,E1 -9407.017,E2 -9407.017} C_VEL
LIN {X 0,Y 432.33,Z 269.255,A -85,B 0,C 180,E1 -9409.822,E2 -9409.822} C_VEL
LIN {X 0,Y 432.299,Z 269.26,A -85,B 0,C 180,E1 -9413.023,E2 -9413.023} C_VEL
LIN {X 0,Y 432.354,Z 269.25,A -85,B 0,C 180,E1 -9415.998,E2 -9415.998} C_VEL
LIN {X 0,Y 432.367,Z 269.335,A -85,B 0,C 180,E1 -9416.519,E2 -9416.519} C_VEL
LIN {X 0,Y 437.214,Z 288.412,A -85,B 0,C 180,E1 -9419.848,E2 -9419.848} C_VEL
LIN {X 0,Y 438.725,Z 295.412,A -85,B 0,C 180,E1 -9421.017,E2 -9421.017} C_VEL
LIN {X 0,Y 437.266,Z 316.195,A -85,B 0,C 180,E1 -9424.086,E2 -9424.086} C_VEL
LIN {X 0,Y 442.543,Z 347.567,A -85,B 0,C 180,E1 -9425.04,E2 -9425.04} C_VEL
LIN {X 0,Y 439.433,Z 483.592,A -85,B 0,C 180,E1 -9427.678,E2 -9427.678} C_VEL
LIN {X 0,Y 438.785,Z 499.51,A -85,B 0,C 180,E1 -9428.169,E2 -9428.169} C_VEL
LIN {X 0,Y 437.984,Z 514.651,A -85,B 0,C 180,E1 -9428.826,E2 -9428.826} C_VEL
LIN {X 0,Y 437.021,Z 529.238,A -85,B 0,C 180,E1 -9429.651,E2 -9429.651} C_VEL
LIN {X 0,Y 436.171,Z 542.525,A -85,B 0,C 180,E1 -9430.591,E2 -9430.591} C_VEL
LIN {X 0,Y 435.11,Z 556.104,A -85,B 0,C 180,E1 -9431.764,E2 -9431.764} C_VEL
LIN {X 0,Y 434.23,Z 568.522,A -85,B 0,C 180,E1 -9433.064,E2 -9433.064} C_VEL
LIN {X 0,Y 433.344,Z 579.855,A -85,B 0,C 180,E1 -9434.48,E2 -9434.48} C_VEL
LIN {X 0,Y 432.733,Z 589.45,A -85,B 0,C 180,E1 -9435.902,E2 -9435.902} C_VEL
LIN {X 0,Y 432.059,Z 598.811,A -85,B 0,C 180,E1 -9437.556,E2 -9437.556} C_VEL
LIN {X 0,Y 431.799,Z 606.562,A -85,B 0,C 180,E1 -9439.213,E2 -9439.213} C_VEL
LIN {X 0,Y 431.453,Z 613.749,A -85,B 0,C 180,E1 -9441.099,E2 -9441.099} C_VEL
LIN {X 0,Y 431.373,Z 619.355,A -85,B 0,C 180,E1 -9442.983,E2 -9442.983} C_VEL
LIN {X 0,Y 431.264,Z 622.589,A -85,B 0,C 180,E1 -9444.39,E2 -9444.39} C_VEL
LIN {X 0,Y 431.235,Z 625.762,A -85,B 0,C 180,E1 -9446.264,E2 -9446.264} C_VEL
LIN {X 0,Y 431.283,Z 627.65,A -85,B 0,C 180,E1 -9448.134,E2 -9448.134} C_VEL
LIN {X 0,Y 431.277,Z 628.245,A -85,B 0,C 180,E1 -9450.001,E2 -9450.001} C_VEL
LIN {X 0,Y 431.287,Z 627.578,A -85,B 0,C 180,E1 -9451.869,E2 -9451.869} C_VEL
LIN {X 0,Y 431.246,Z 625.66,A -85,B 0,C 180,E1 -9453.739,E2 -9453.739} C_VEL
LIN {X 0,Y 431.299,Z 622.466,A -85,B 0,C 180,E1 -9455.612,E2 -9455.612} C_VEL
LIN {X 0,Y 431.346,Z 617.914,A -85,B 0,C 180,E1 -9457.491,E2 -9457.491} C_VEL
LIN {X 0,Y 431.497,Z 611.906,A -85,B 0,C 180,E1 -9459.375,E2 -9459.375} C_VEL
LIN {X 0,Y 431.872,Z 604.272,A -85,B 0,C 180,E1 -9461.262,E2 -9461.262} C_VEL
LIN {X 0,Y 432.286,Z 595.816,A -85,B 0,C 180,E1 -9462.97,E2 -9462.97} C_VEL
LIN {X 0,Y 432.896,Z 586.272,A -85,B 0,C 180,E1 -9464.576,E2 -9464.576} C_VEL
LIN {X 0,Y 433.641,Z 576.282,A -85,B 0,C 180,E1 -9465.994,E2 -9465.994} C_VEL
LIN {X 0,Y 434.538,Z 564.542,A -85,B 0,C 180,E1 -9467.4,E2 -9467.4} C_VEL
LIN {X 0,Y 435.481,Z 551.471,A -85,B 0,C 180,E1 -9468.71,E2 -9468.71} C_VEL
LIN {X 0,Y 436.625,Z 537.224,A -85,B 0,C 180,E1 -9469.88,E2 -9469.88} C_VEL
LIN {X 0,Y 437.657,Z 523.543,A -85,B 0,C 180,E1 -9470.8,E2 -9470.8} C_VEL
LIN {X 0,Y 438.674,Z 508.216,A -85,B 0,C 180,E1 -9471.623,E2 -9471.623} C_VEL
LIN {X 0,Y 439.556,Z 492.691,A -85,B 0,C 180,E1 -9472.256,E2 -9472.256} C_VEL
LIN {X 0,Y 440.357,Z 476.906,A -85,B 0,C 180,E1 -9472.709,E2 -9472.709} C_VEL
LIN {X 0,Y 443.172,Z 388.54,A -85,B 0,C 180,E1 -9474.608,E2 -9474.608} C_VEL
LIN {X 0,Y 444.654,Z 347.098,A -85,B 0,C 180,E1 -9475.567,E2 -9475.567} C_VEL
LIN {X 0,Y 442.302,Z 330.015,A -85,B 0,C 180,E1 -9476.23,E2 -9476.23} C_VEL
LIN {X 0,Y 439.118,Z 313.559,A -85,B 0,C 180,E1 -9476.986,E2 -9476.986} C_VEL
LIN {X 0,Y 438.397,Z 310.019,A -85,B 0,C 180,E1 -9477.187,E2 -9477.187} C_VEL
LIN {X 0,Y 439.738,Z 297.802,A -85,B 0,C 180,E1 -9479.175,E2 -9479.175} C_VEL
LIN {X 0,Y 438.781,Z 291.639,A -85,B 0,C 180,E1 -9480.38,E2 -9480.38} C_VEL
LIN {X 0,Y 436.155,Z 281.298,A -85,B 0,C 180,E1 -9482.669,E2 -9482.669} C_VEL
LIN {X 0,Y 433.833,Z 273.993,A -85,B 0,C 180,E1 -9484.542,E2 -9484.542} C_VEL
LIN {X 0,Y 432.352,Z 269.257,A -85,B 0,C 180,E1 -9485.889,E2 -9485.889} C_VEL
LIN {X 0,Y 432.355,Z 269.256,A -85,B 0,C 180,E1 -9489.343,E2 -9489.343} C_VEL
LIN {X 0,Y 432.34,Z 269.257,A -85,B 0,C 180,E1 -9491.798,E2 -9491.798} C_VEL
LIN {X 0,Y 432.34,Z 269.257,A -85,B 0,C 180,E1 -9494.348,E2 -9494.348} C_VEL
LIN {X 0,Y 432.327,Z 269.26,A -85,B 0,C 180,E1 -9497.016,E2 -9497.016} C_VEL
LIN {X 0,Y 432.34,Z 269.255,A -85,B 0,C 180,E1 -9499.821,E2 -9499.821} C_VEL
LIN {X 0,Y 432.311,Z 269.261,A -85,B 0,C 180,E1 -9503.022,E2 -9503.022} C_VEL
LIN {X 0,Y 432.366,Z 269.254,A -85,B 0,C 180,E1 -9505.997,E2 -9505.997} C_VEL
LIN {X 0,Y 432.353,Z 269.257,A -85,B 0,C 180,E1 -9509.49,E2 -9509.49} C_VEL
LIN {X 0,Y 432.361,Z 269.307,A -85,B 0,C 180,E1 -9510.077,E2 -9510.077} C_VEL
LIN {X 0,Y 434.724,Z 277.093,A -85,B 0,C 180,E1 -9512.573,E2 -9512.573} C_VEL
LIN {X 0,Y 441.181,Z 288.643,A -85,B 0,C 180,E1 -9513.591,E2 -9513.591} C_VEL
LIN {X 0,Y 445.801,Z 298.232,A -85,B 0,C 180,E1 -9514.291,E2 -9514.291} C_VEL
LIN {X 0,Y 445.975,Z 300.069,A -85,B 0,C 180,E1 -9514.358,E2 -9514.358} C_VEL
LIN {X 0,Y 442.369,Z 386.834,A -85,B 0,C 180,E1 -9516.349,E2 -9516.349} C_VEL
LIN {X 0,Y 440.766,Z 439.271,A -85,B 0,C 180,E1 -9517.5,E2 -9517.5} C_VEL
LIN {X 0,Y 440.106,Z 455.238,A -85,B 0,C 180,E1 -9518.037,E2 -9518.037} C_VEL
LIN {X 0,Y 439.378,Z 469.93,A -85,B 0,C 180,E1 -9518.721,E2 -9518.721} C_VEL
LIN {X 0,Y 438.542,Z 484.53,A -85,B 0,C 180,E1 -9519.6,E2 -9519.6} C_VEL
LIN {X 0,Y 437.573,Z 498.57,A -85,B 0,C 180,E1 -9520.654,E2 -9520.654} C_VEL
LIN {X 0,Y 436.463,Z 511.871,A -85,B 0,C 180,E1 -9521.872,E2 -9521.872} C_VEL
LIN {X 0,Y 435.503,Z 523.103,A -85,B 0,C 180,E1 -9523.113,E2 -9523.113} C_VEL
LIN {X 0,Y 434.688,Z 533.823,A -85,B 0,C 180,E1 -9524.527,E2 -9524.527} C_VEL
LIN {X 0,Y 433.725,Z 544.253,A -85,B 0,C 180,E1 -9526.17,E2 -9526.17} C_VEL
LIN {X 0,Y 433.138,Z 551.759,A -85,B 0,C 180,E1 -9527.584,E2 -9527.584} C_VEL
LIN {X 0,Y 432.55,Z 559.108,A -85,B 0,C 180,E1 -9529.23,E2 -9529.23} C_VEL
LIN {X 0,Y 432.08,Z 565.859,A -85,B 0,C 180,E1 -9531.11,E2 -9531.11} C_VEL
LIN {X 0,Y 431.843,Z 569.895,A -85,B 0,C 180,E1 -9532.518,E2 -9532.518} C_VEL
LIN {X 0,Y 431.528,Z 574.095,A -85,B 0,C 180,E1 -9534.392,E2 -9534.392} C_VEL
LIN {X 0,Y 431.491,Z 576.983,A -85,B 0,C 180,E1 -9536.264,E2 -9536.264} C_VEL
LIN {X 0,Y 431.394,Z 578.653,A -85,B 0,C 180,E1 -9538.132,E2 -9538.132} C_VEL
LIN {X 0,Y 431.281,Z 579.128,A -85,B 0,C 180,E1 -9539.999,E2 -9539.999} C_VEL
LIN {X 0,Y 431.334,Z 578.365,A -85,B 0,C 180,E1 -9541.867,E2 -9541.867} C_VEL
LIN {X 0,Y 431.45,Z 576.379,A -85,B 0,C 180,E1 -9543.735,E2 -9543.735} C_VEL
LIN {X 0,Y 431.522,Z 573.159,A -85,B 0,C 180,E1 -9545.607,E2 -9545.607} C_VEL
LIN {X 0,Y 431.691,Z 568.624,A -85,B 0,C 180,E1 -9547.483,E2 -9547.483} C_VEL
LIN {X 0,Y 431.966,Z 562.663,A -85,B 0,C 180,E1 -9549.363,E2 -9549.363} C_VEL
LIN {X 0,Y 432.445,Z 555.1,A -85,B 0,C 180,E1 -9551.245,E2 -9551.245} C_VEL
LIN {X 0,Y 432.989,Z 546.648,A -85,B 0,C 180,E1 -9552.954,E2 -9552.954} C_VEL
LIN {X 0,Y 433.664,Z 537.15,A -85,B 0,C 180,E1 -9554.547,E2 -9554.547} C_VEL
LIN {X 0,Y 434.444,Z 527.104,A -85,B 0,C 180,E1 -9555.962,E2 -9555.962} C_VEL
LIN {X 0,Y 435.317,Z 515.527,A -85,B 0,C 180,E1 -9557.333,E2 -9557.333} C_VEL
LIN {X 0,Y 436.167,Z 503.202,A -85,B 0,C 180,E1 -9558.555,E2 -9558.555} C_VEL
LIN {X 0,Y 437.051,Z 490.35,A -85,B 0,C 180,E1 -9559.613,E2 -9559.613} C_VEL
LIN {X 0,Y 437.904,Z 476.373,A -85,B 0,C 180,E1 -9560.552,E2 -9560.552} C_VEL
LIN {X 0,Y 438.663,Z 462.1,A -85,B 0,C 180,E1 -9561.313,E2 -9561.313} C_VEL
LIN {X 0,Y 439.204,Z 447.107,A -85,B 0,C 180,E1 -9561.926,E2 -9561.926} C_VEL
LIN {X 0,Y 439.727,Z 431.849,A -85,B 0,C 180,E1 -9562.36,E2 -9562.36} C_VEL
LIN {X 0,Y 442.752,Z 295.324,A -85,B 0,C 180,E1 -9565.002,E2 -9565.002} C_VEL
LIN {X 0,Y 433.044,Z 271.52,A -85,B 0,C 180,E1 -9566.049,E2 -9566.049} C_VEL
LIN {X 0,Y 432.372,Z 269.253,A -85,B 0,C 180,E1 -9566.161,E2 -9566.161} C_VEL
LIN {X 0,Y 432.334,Z 269.255,A -85,B 0,C 180,E1 -9569.187,E2 -9569.187} C_VEL
LIN {X 0,Y 432.324,Z 269.257,A -85,B 0,C 180,E1 -9572.442,E2 -9572.442} C_VEL
LIN {X 0,Y 432.343,Z 269.256,A -85,B 0,C 180,E1 -9575.63,E2 -9575.63} C_VEL
LIN {X 0,Y 432.325,Z 269.253,A -85,B 0,C 180,E1 -9578.711,E2 -9578.711} C_VEL
LIN {X 0,Y 432.323,Z 269.261,A -85,B 0,C 180,E1 -9581.797,E2 -9581.797} C_VEL
LIN {X 0,Y 432.332,Z 269.254,A -85,B 0,C 180,E1 -9584.346,E2 -9584.346} C_VEL
LIN {X 0,Y 432.318,Z 269.254,A -85,B 0,C 180,E1 -9587.014,E2 -9587.014} C_VEL
LIN {X 0,Y 432.331,Z 269.26,A -85,B 0,C 180,E1 -9589.819,E2 -9589.819} C_VEL
LIN {X 0,Y 432.303,Z 269.256,A -85,B 0,C 180,E1 -9593.021,E2 -9593.021} C_VEL
LIN {X 0,Y 432.354,Z 269.254,A -85,B 0,C 180,E1 -9595.996,E2 -9595.996} C_VEL
LIN {X 0,Y 432.342,Z 269.256,A -85,B 0,C 180,E1 -9599.489,E2 -9599.489} C_VEL
LIN {X 0,Y 432.343,Z 269.257,A -85,B 0,C 180,E1 -9601.873,E2 -9601.873} C_VEL
LIN {X 0,Y 432.374,Z 269.253,A -85,B 0,C 180,E1 -9605.537,E2 -9605.537} C_VEL
LIN {X 0,Y 432.344,Z 269.252,A -85,B 0,C 180,E1 -9609.045,E2 -9609.045} C_VEL
LIN {X 0,Y 432.353,Z 269.25,A -85,B 0,C 180,E1 -9611.442,E2 -9611.442} C_VEL
LIN {X 0,Y 431.671,Z 269.338,A -85,B 0,C 180,E1 -9612.22,E2 -9612.22} C_VEL
LIN {X 0,Y 428.807,Z 269.697,A -85,B 0,C 180,E1 -9613.483,E2 -9613.483} C_VEL
LIN {X 0,Y 426.408,Z 269.992,A -85,B 0,C 180,E1 -9614.503,E2 -9614.503} C_VEL
LIN {X 0,Y 425.405,Z 270.119,A -85,B 0,C 180,E1 -9615.291,E2 -9615.291} C_VEL
LIN {X 0,Y 425.336,Z 270.13,A -85,B 0,C 180,E1 -9615.558,E2 -9615.558} C_VEL
LIN {X 0,Y 425.344,Z 270.123,A -85,B 0,C 180,E1 -9618.563,E2 -9618.563} C_VEL
LIN {X 0,Y 425.531,Z 270.1,A -85,B 0,C 180,E1 -9622.406,E2 -9622.406} C_VEL
LIN {X 0,Y 425.542,Z 270.099,A -85,B 0,C 180,E1 -9624.312,E2 -9624.312} C_VEL
LIN {X 0,Y 425.564,Z 270.097,A -85,B 0,C 180,E1 -9628.106,E2 -9628.106} C_VEL
LIN {X 0,Y 425.694,Z 270.082,A -85,B 0,C 180,E1 -9629.999,E2 -9629.999} C_VEL
LIN {X 0,Y 425.537,Z 270.1,A -85,B 0,C 180,E1 -9632.839,E2 -9632.839} C_VEL
LIN {X 0,Y 425.518,Z 270.101,A -85,B 0,C 180,E1 -9636.638,E2 -9636.638} C_VEL
LIN {X 0,Y 425.39,Z 270.125,A -85,B 0,C 180,E1 -9639.508,E2 -9639.508} C_VEL
LIN {X 0,Y 425.383,Z 270.12,A -85,B 0,C 180,E1 -9642.902,E2 -9642.902} C_VEL
LIN {X 0,Y 425.35,Z 270.122,A -85,B 0,C 180,E1 -9646.604,E2 -9646.604} C_VEL
LIN {X 0,Y 425.317,Z 270.131,A -85,B 0,C 180,E1 -9649.635,E2 -9649.635} C_VEL
LIN {X 0,Y 425.292,Z 270.137,A -85,B 0,C 180,E1 -9653.364,E2 -9653.364} C_VEL
LIN {X 0,Y 425.335,Z 270.126,A -85,B 0,C 180,E1 -9656.843,E2 -9656.843} C_VEL
LIN {X 0,Y 425.278,Z 270.135,A -85,B 0,C 180,E1 -9659.719,E2 -9659.719} C_VEL
LIN {X 0,Y 425.269,Z 270.136,A -85,B 0,C 180,E1 -9663.047,E2 -9663.047} C_VEL
LIN {X 0,Y 425.27,Z 270.133,A -85,B 0,C 180,E1 -9665.928,E2 -9665.928} C_VEL
LIN {X 0,Y 425.286,Z 270.134,A -85,B 0,C 180,E1 -9669.043,E2 -9669.043} C_VEL
LIN {X 0,Y 425.264,Z 270.134,A -85,B 0,C 180,E1 -9672.652,E2 -9672.652} C_VEL
LIN {X 0,Y 425.254,Z 270.135,A -85,B 0,C 180,E1 -9676.045,E2 -9676.045} C_VEL
LIN {X 0,Y 425.261,Z 270.134,A -85,B 0,C 180,E1 -9678.621,E2 -9678.621} C_VEL
LIN {X 0,Y 425.291,Z 270.135,A -85,B 0,C 180,E1 -9681.102,E2 -9681.102} C_VEL
LIN {X 0,Y 425.285,Z 270.132,A -85,B 0,C 180,E1 -9684.664,E2 -9684.664} C_VEL
LIN {X 0,Y 425.25,Z 270.135,A -85,B 0,C 180,E1 -9688.073,E2 -9688.073} C_VEL
LIN {X 0,Y 425.316,Z 270.132,A -85,B 0,C 180,E1 -9691.368,E2 -9691.368} C_VEL
LIN {X 0,Y 425.28,Z 270.132,A -85,B 0,C 180,E1 -9694.555,E2 -9694.555} C_VEL
LIN {X 0,Y 425.273,Z 270.134,A -85,B 0,C 180,E1 -9697.661,E2 -9697.661} C_VEL
LIN {X 0,Y 425.347,Z 270.125,A -85,B 0,C 180,E1 -9700.704,E2 -9700.704} C_VEL
LIN {X 0,Y 425.374,Z 270.121,A -85,B 0,C 180,E1 -9703.689,E2 -9703.689} C_VEL
LIN {X 0,Y 425.398,Z 270.118,A -85,B 0,C 180,E1 -9707.599,E2 -9707.599} C_VEL
LIN {X 0,Y 425.428,Z 270.115,A -85,B 0,C 180,E1 -9711.45,E2 -9711.45} C_VEL
LIN {X 0,Y 425.535,Z 270.1,A -85,B 0,C 180,E1 -9714.314,E2 -9714.314} C_VEL
LIN {X 0,Y 425.563,Z 270.096,A -85,B 0,C 180,E1 -9718.108,E2 -9718.108} C_VEL
LIN {X 0,Y 425.689,Z 270.08,A -85,B 0,C 180,E1 -9720.001,E2 -9720.001} C_VEL
LIN {X 0,Y 425.532,Z 270.105,A -85,B 0,C 180,E1 -9722.841,E2 -9722.841} C_VEL
LIN {X 0,Y 425.515,Z 270.105,A -85,B 0,C 180,E1 -9726.64,E2 -9726.64} C_VEL
LIN {X 0,Y 425.389,Z 270.119,A -85,B 0,C 180,E1 -9729.51,E2 -9729.51} C_VEL
LIN {X 0,Y 425.381,Z 270.126,A -85,B 0,C 180,E1 -9732.905,E2 -9732.905} C_VEL
LIN {X 0,Y 425.35,Z 270.126,A -85,B 0,C 180,E1 -9736.606,E2 -9736.606} C_VEL
LIN {X 0,Y 425.318,Z 270.127,A -85,B 0,C 180,E1 -9739.637,E2 -9739.637} C_VEL
LIN {X 0,Y 425.277,Z 270.133,A -85,B 0,C 180,E1 -9742.34,E2 -9742.34} C_VEL
LIN {X 0,Y 425.282,Z 270.132,A -85,B 0,C 180,E1 -9745.447,E2 -9745.447} C_VEL
LIN {X 0,Y 425.321,Z 270.131,A -85,B 0,C 180,E1 -9748.633,E2 -9748.633} C_VEL
LIN {X 0,Y 425.255,Z 270.134,A -85,B 0,C 180,E1 -9751.928,E2 -9751.928} C_VEL
LIN {X 0,Y 425.29,Z 270.131,A -85,B 0,C 180,E1 -9755.337,E2 -9755.337} C_VEL
LIN {X 0,Y 425.29,Z 270.136,A -85,B 0,C 180,E1 -9758.9,E2 -9758.9} C_VEL
LIN {X 0,Y 425.282,Z 270.131,A -85,B 0,C 180,E1 -9761.96,E2 -9761.96} C_VEL
LIN {X 0,Y 425.278,Z 270.133,A -85,B 0,C 180,E1 -9765.285,E2 -9765.285} C_VEL
LIN {X 0,Y 425.268,Z 270.139,A -85,B 0,C 180,E1 -9768.623,E2 -9768.623} C_VEL
LIN {X 0,Y 425.303,Z 270.133,A -85,B 0,C 180,E1 -9771.104,E2 -9771.104} C_VEL
LIN {X 0,Y 425.293,Z 270.132,A -85,B 0,C 180,E1 -9774.666,E2 -9774.666} C_VEL
LIN {X 0,Y 425.335,Z 270.271,A -85,B 0,C 180,E1 -9776.179,E2 -9776.179} C_VEL
LIN {X 0,Y 430.164,Z 289.382,A -85,B 0,C 180,E1 -9779.572,E2 -9779.572} C_VEL
LIN {X 0,Y 431.81,Z 296.425,A -85,B 0,C 180,E1 -9780.775,E2 -9780.775} C_VEL
LIN {X 0,Y 431.016,Z 308.338,A -85,B 0,C 180,E1 -9782.574,E2 -9782.574} C_VEL
LIN {X 0,Y 430.492,Z 316.252,A -85,B 0,C 180,E1 -9783.718,E2 -9783.718} C_VEL
LIN {X 0,Y 435.931,Z 348.149,A -85,B 0,C 180,E1 -9784.707,E2 -9784.707} C_VEL
LIN {X 0,Y 432.966,Z 474.543,A -85,B 0,C 180,E1 -9787.2,E2 -9787.2} C_VEL
LIN {X 0,Y 432.376,Z 491.02,A -85,B 0,C 180,E1 -9787.608,E2 -9787.608} C_VEL
LIN {X 0,Y 431.578,Z 506.962,A -85,B 0,C 180,E1 -9788.209,E2 -9788.209} C_VEL
LIN {X 0,Y 430.68,Z 521.778,A -85,B 0,C 180,E1 -9788.963,E2 -9788.963} C_VEL
LIN {X 0,Y 429.778,Z 534.767,A -85,B 0,C 180,E1 -9789.792,E2 -9789.792} C_VEL
LIN {X 0,Y 428.783,Z 548.391,A -85,B 0,C 180,E1 -9790.866,E2 -9790.866} C_VEL
LIN {X 0,Y 427.846,Z 560.498,A -85,B 0,C 180,E1 -9792.018,E2 -9792.018} C_VEL
LIN {X 0,Y 426.946,Z 571.494,A -85,B 0,C 180,E1 -9793.259,E2 -9793.259} C_VEL
LIN {X 0,Y 426.125,Z 582.296,A -85,B 0,C 180,E1 -9794.701,E2 -9794.701} C_VEL
LIN {X 0,Y 425.533,Z 591.44,A -85,B 0,C 180,E1 -9796.146,E2 -9796.146} C_VEL
LIN {X 0,Y 424.966,Z 600.409,A -85,B 0,C 180,E1 -9797.829,E2 -9797.829} C_VEL
LIN {X 0,Y 424.622,Z 607.841,A -85,B 0,C 180,E1 -9799.511,E2 -9799.511} C_VEL
LIN {X 0,Y 424.357,Z 614.679,A -85,B 0,C 180,E1 -9801.429,E2 -9801.429} C_VEL
LIN {X 0,Y 424.237,Z 619.974,A -85,B 0,C 180,E1 -9803.342,E2 -9803.342} C_VEL
LIN {X 0,Y 424.169,Z 623.857,A -85,B 0,C 180,E1 -9805.249,E2 -9805.249} C_VEL
LIN {X 0,Y 424.243,Z 626.421,A -85,B 0,C 180,E1 -9807.153,E2 -9807.153} C_VEL
LIN {X 0,Y 424.201,Z 627.676,A -85,B 0,C 180,E1 -9809.052,E2 -9809.052} C_VEL
LIN {X 0,Y 424.189,Z 627.652,A -85,B 0,C 180,E1 -9810.951,E2 -9810.951} C_VEL
LIN {X 0,Y 424.258,Z 626.378,A -85,B 0,C 180,E1 -9812.85,E2 -9812.85} C_VEL
LIN {X 0,Y 424.186,Z 623.834,A -85,B 0,C 180,E1 -9814.753,E2 -9814.753} C_VEL
LIN {X 0,Y 424.219,Z 619.981,A -85,B 0,C 180,E1 -9816.661,E2 -9816.661} C_VEL
LIN {X 0,Y 424.356,Z 614.716,A -85,B 0,C 180,E1 -9818.573,E2 -9818.573} C_VEL
LIN {X 0,Y 424.604,Z 607.924,A -85,B 0,C 180,E1 -9820.492,E2 -9820.492} C_VEL
LIN {X 0,Y 424.969,Z 600.592,A -85,B 0,C 180,E1 -9822.174,E2 -9822.174} C_VEL
LIN {X 0,Y 425.547,Z 591.766,A -85,B 0,C 180,E1 -9823.856,E2 -9823.856} C_VEL
LIN {X 0,Y 426.3,Z 581.129,A -85,B 0,C 180,E1 -9825.54,E2 -9825.54} C_VEL
LIN {X 0,Y 427.098,Z 570.303,A -85,B 0,C 180,E1 -9826.984,E2 -9826.984} C_VEL
LIN {X 0,Y 428.246,Z 557.372,A -85,B 0,C 180,E1 -9828.417,E2 -9828.417} C_VEL
LIN {X 0,Y 429.319,Z 544.513,A -85,B 0,C 180,E1 -9829.609,E2 -9829.609} C_VEL
LIN {X 0,Y 430.432,Z 530.551,A -85,B 0,C 180,E1 -9830.677,E2 -9830.677} C_VEL
LIN {X 0,Y 431.619,Z 514.977,A -85,B 0,C 180,E1 -9831.634,E2 -9831.634} C_VEL
LIN {X 0,Y 432.658,Z 499.456,A -85,B 0,C 180,E1 -9832.372,E2 -9832.372} C_VEL
LIN {X 0,Y 433.626,Z 483.592,A -85,B 0,C 180,E1 -9832.924,E2 -9832.924} C_VEL
LIN {X 0,Y 434.474,Z 459.917,A -85,B 0,C 180,E1 -9833.475,E2 -9833.475} C_VEL
LIN {X 0,Y 437.358,Z 379.776,A -85,B 0,C 180,E1 -9835.277,E2 -9835.277} C_VEL
LIN {X 0,Y 438.641,Z 348.433,A -85,B 0,C 180,E1 -9836.029,E2 -9836.029} C_VEL
LIN {X 0,Y 436.529,Z 332.213,A -85,B 0,C 180,E1 -9836.681,E2 -9836.681} C_VEL
LIN {X 0,Y 433.389,Z 315.672,A -85,B 0,C 180,E1 -9837.477,E2 -9837.477} C_VEL
LIN {X 0,Y 432.083,Z 309.329,A -85,B 0,C 180,E1 -9837.831,E2 -9837.831} C_VEL
LIN {X 0,Y 433.202,Z 300.008,A -85,B 0,C 180,E1 -9839.391,E2 -9839.391} C_VEL
LIN {X 0,Y 432.011,Z 292.974,A -85,B 0,C 180,E1 -9840.827,E2 -9840.827} C_VEL
LIN {X 0,Y 429.573,Z 283.457,A -85,B 0,C 180,E1 -9843.035,E2 -9843.035} C_VEL
LIN {X 0,Y 427.128,Z 275.612,A -85,B 0,C 180,E1 -9845.163,E2 -9845.163} C_VEL
LIN {X 0,Y 425.276,Z 270.138,A -85,B 0,C 180,E1 -9846.915,E2 -9846.915} C_VEL
LIN {X 0,Y 425.296,Z 270.135,A -85,B 0,C 180,E1 -9850.127,E2 -9850.127} C_VEL
LIN {X 0,Y 425.264,Z 270.139,A -85,B 0,C 180,E1 -9853.351,E2 -9853.351} C_VEL
LIN {X 0,Y 425.264,Z 270.138,A -85,B 0,C 180,E1 -9856.649,E2 -9856.649} C_VEL
LIN {X 0,Y 425.293,Z 270.133,A -85,B 0,C 180,E1 -9859.873,E2 -9859.873} C_VEL
LIN {X 0,Y 425.283,Z 270.138,A -85,B 0,C 180,E1 -9862.489,E2 -9862.489} C_VEL
LIN {X 0,Y 425.314,Z 270.133,A -85,B 0,C 180,E1 -9865.817,E2 -9865.817} C_VEL
LIN {X 0,Y 425.328,Z 270.321,A -85,B 0,C 180,E1 -9869.118,E2 -9869.118} C_VEL
LIN {X 0,Y 427.474,Z 277.148,A -85,B 0,C 180,E1 -9871.524,E2 -9871.524} C_VEL
LIN {X 0,Y 427.879,Z 278.29,A -85,B 0,C 180,E1 -9871.841,E2 -9871.841} C_VEL
LIN {X 0,Y 434.683,Z 290.007,A -85,B 0,C 180,E1 -9872.983,E2 -9872.983} C_VEL
LIN {X 0,Y 439.814,Z 300.342,A -85,B 0,C 180,E1 -9873.805,E2 -9873.805} C_VEL
LIN {X 0,Y 440.025,Z 302.473,A -85,B 0,C 180,E1 -9873.887,E2 -9873.887} C_VEL
LIN {X 0,Y 436.179,Z 387.093,A -85,B 0,C 180,E1 -9875.898,E2 -9875.898} C_VEL
LIN {X 0,Y 434.386,Z 440.536,A -85,B 0,C 180,E1 -9877.119,E2 -9877.119} C_VEL
LIN {X 0,Y 433.659,Z 456.468,A -85,B 0,C 180,E1 -9877.676,E2 -9877.676} C_VEL
LIN {X 0,Y 432.797,Z 472.264,A -85,B 0,C 180,E1 -9878.444,E2 -9878.444} C_VEL
LIN {X 0,Y 431.868,Z 487.293,A -85,B 0,C 180,E1 -9879.395,E2 -9879.395} C_VEL
LIN {X 0,Y 430.804,Z 500.881,A -85,B 0,C 180,E1 -9880.462,E2 -9880.462} C_VEL
LIN {X 0,Y 429.761,Z 512.807,A -85,B 0,C 180,E1 -9881.592,E2 -9881.592} C_VEL
LIN {X 0,Y 428.751,Z 523.847,A -85,B 0,C 180,E1 -9882.839,E2 -9882.839} C_VEL
LIN {X 0,Y 427.872,Z 534.517,A -85,B 0,C 180,E1 -9884.274,E2 -9884.274} C_VEL
LIN {X 0,Y 426.969,Z 543.557,A -85,B 0,C 180,E1 -9885.705,E2 -9885.705} C_VEL
LIN {X 0,Y 426.195,Z 552.379,A -85,B 0,C 180,E1 -9887.379,E2 -9887.379} C_VEL
LIN {X 0,Y 425.586,Z 559.694,A -85,B 0,C 180,E1 -9889.052,E2 -9889.052} C_VEL
LIN {X 0,Y 425.083,Z 566.416,A -85,B 0,C 180,E1 -9890.963,E2 -9890.963} C_VEL
LIN {X 0,Y 424.8,Z 570.44,A -85,B 0,C 180,E1 -9892.394,E2 -9892.394} C_VEL
LIN {X 0,Y 424.484,Z 574.609,A -85,B 0,C 180,E1 -9894.298,E2 -9894.298} C_VEL
LIN {X 0,Y 424.431,Z 577.467,A -85,B 0,C 180,E1 -9896.202,E2 -9896.202} C_VEL
LIN {X 0,Y 424.311,Z 579.107,A -85,B 0,C 180,E1 -9898.101,E2 -9898.101} C_VEL
LIN {X 0,Y 424.207,Z 579.542,A -85,B 0,C 180,E1 -9899.999,E2 -9899.999} C_VEL
LIN {X 0,Y 424.255,Z 578.75,A -85,B 0,C 180,E1 -9901.898,E2 -9901.898} C_VEL
LIN {X 0,Y 424.355,Z 576.719,A -85,B 0,C 180,E1 -9903.798,E2 -9903.798} C_VEL
LIN {X 0,Y 424.452,Z 573.442,A -85,B 0,C 180,E1 -9905.701,E2 -9905.701} C_VEL
LIN {X 0,Y 424.633,Z 568.844,A -85,B 0,C 180,E1 -9907.608,E2 -9907.608} C_VEL
LIN {X 0,Y 424.942,Z 562.811,A -85,B 0,C 180,E1 -9909.519,E2 -9909.519} C_VEL
LIN {X 0,Y 425.469,Z 555.167,A -85,B 0,C 180,E1 -9911.432,E2 -9911.432} C_VEL
LIN {X 0,Y 425.991,Z 547.107,A -85,B 0,C 180,E1 -9913.078,E2 -9913.078} C_VEL
LIN {X 0,Y 426.737,Z 537.019,A -85,B 0,C 180,E1 -9914.789,E2 -9914.789} C_VEL
LIN {X 0,Y 427.534,Z 526.85,A -85,B 0,C 180,E1 -9916.227,E2 -9916.227} C_VEL
LIN {X 0,Y 428.434,Z 515.591,A -85,B 0,C 180,E1 -9917.569,E2 -9917.569} C_VEL
LIN {X 0,Y 429.353,Z 502.632,A -85,B 0,C 180,E1 -9918.861,E2 -9918.861} C_VEL
LIN {X 0,Y 430.29,Z 489.568,A -85,B 0,C 180,E1 -9919.934,E2 -9919.934} C_VEL
LIN {X 0,Y 431.128,Z 475.299,A -85,B 0,C 180,E1 -9920.89,E2 -9920.89} C_VEL
LIN {X 0,Y 431.939,Z 460.633,A -85,B 0,C 180,E1 -9921.662,E2 -9921.662} C_VEL
LIN {X 0,Y 432.558,Z 445.287,A -85,B 0,C 180,E1 -9922.272,E2 -9922.272} C_VEL
LIN {X 0,Y 433.022,Z 429.473,A -85,B 0,C 180,E1 -9922.703,E2 -9922.703} C_VEL
LIN {X 0,Y 436.142,Z 296.989,A -85,B 0,C 180,E1 -9925.324,E2 -9925.324} C_VEL
LIN {X 0,Y 426.324,Z 273.004,A -85,B 0,C 180,E1 -9926.399,E2 -9926.399} C_VEL
LIN {X 0,Y 425.314,Z 270.131,A -85,B 0,C 180,E1 -9926.527,E2 -9926.527} C_VEL
LIN {X 0,Y 425.287,Z 270.136,A -85,B 0,C 180,E1 -9929.719,E2 -9929.719} C_VEL
LIN {X 0,Y 425.283,Z 270.131,A -85,B 0,C 180,E1 -9933.047,E2 -9933.047} C_VEL
LIN {X 0,Y 425.281,Z 270.138,A -85,B 0,C 180,E1 -9935.927,E2 -9935.927} C_VEL
LIN {X 0,Y 425.261,Z 270.133,A -85,B 0,C 180,E1 -9939.036,E2 -9939.036} C_VEL
LIN {X 0,Y 425.281,Z 270.137,A -85,B 0,C 180,E1 -9941.956,E2 -9941.956} C_VEL
LIN {X 0,Y 425.283,Z 270.132,A -85,B 0,C 180,E1 -9945.282,E2 -9945.282} C_VEL
LIN {X 0,Y 425.271,Z 270.132,A -85,B 0,C 180,E1 -9948.62,E2 -9948.62} C_VEL
LIN {X 0,Y 425.294,Z 270.13,A -85,B 0,C 180,E1 -9951.1,E2 -9951.1} C_VEL
LIN {X 0,Y 425.295,Z 270.129,A -85,B 0,C 180,E1 -9954.663,E2 -9954.663} C_VEL
LIN {X 0,Y 425.26,Z 270.137,A -85,B 0,C 180,E1 -9958.072,E2 -9958.072} C_VEL
LIN {X 0,Y 425.31,Z 270.13,A -85,B 0,C 180,E1 -9961.365,E2 -9961.365} C_VEL
LIN {X 0,Y 425.267,Z 270.133,A -85,B 0,C 180,E1 -9964.552,E2 -9964.552} C_VEL
LIN {X 0,Y 425.279,Z 270.131,A -85,B 0,C 180,E1 -9966.632,E2 -9966.632} C_VEL
LIN {X 0,Y 425.29,Z 270.137,A -85,B 0,C 180,E1 -9969.693,E2 -9969.693} C_VEL
LIN {X 0,Y 425.328,Z 270.125,A -85,B 0,C 180,E1 -9972.696,E2 -9972.696} C_VEL
LIN {X 0,Y 425.336,Z 270.13,A -85,B 0,C 180,E1 -9975.558,E2 -9975.558} C_VEL
LIN {X 0,Y 424.705,Z 270.217,A -85,B 0,C 180,E1 -9976.349,E2 -9976.349} C_VEL
LIN {X 0,Y 421.863,Z 270.572,A -85,B 0,C 180,E1 -9977.633,E2 -9977.633} C_VEL
LIN {X 0,Y 419.438,Z 270.867,A -85,B 0,C 180,E1 -9978.671,E2 -9978.671} C_VEL
LIN {X 0,Y 418.398,Z 270.994,A -85,B 0,C 180,E1 -9979.472,E2 -9979.472} C_VEL
LIN {X 0,Y 418.315,Z 270.999,A -85,B 0,C 180,E1 -9979.744,E2 -9979.744} C_VEL
LIN {X 0,Y 418.506,Z 270.976,A -85,B 0,C 180,E1 -9982.278,E2 -9982.278} C_VEL
LIN {X 0,Y 418.501,Z 270.976,A -85,B 0,C 180,E1 -9984.216,E2 -9984.216} C_VEL
LIN {X 0,Y 418.533,Z 270.973,A -85,B 0,C 180,E1 -9988.074,E2 -9988.074} C_VEL
LIN {X 0,Y 418.663,Z 270.958,A -85,B 0,C 180,E1 -9989.999,E2 -9989.999} C_VEL
LIN {X 0,Y 418.492,Z 270.977,A -85,B 0,C 180,E1 -9992.886,E2 -9992.886} C_VEL
LIN {X 0,Y 418.481,Z 270.978,A -85,B 0,C 180,E1 -9996.75,E2 -9996.75} C_VEL
LIN {X 0,Y 418.39,Z 270.989,A -85,B 0,C 180,E1 -9998.694,E2 -9998.694} C_VEL
LIN {X 0,Y 418.305,Z 271.006,A -85,B 0,C 180,E1 -10001.63,E2 -10001.63} C_VEL
LIN {X 0,Y 418.291,Z 271.002,A -85,B 0,C 180,E1 -10004.596,E2 -10004.596} C_VEL
LIN {X 0,Y 418.276,Z 271.009,A -85,B 0,C 180,E1 -10007.603,E2 -10007.603} C_VEL
LIN {X 0,Y 418.238,Z 271.009,A -85,B 0,C 180,E1 -10010.662,E2 -10010.662} C_VEL
LIN {X 0,Y 418.273,Z 271.007,A -85,B 0,C 180,E1 -10013.78,E2 -10013.78} C_VEL
LIN {X 0,Y 418.297,Z 271.004,A -85,B 0,C 180,E1 -10017.07,E2 -10017.07} C_VEL
LIN {X 0,Y 418.231,Z 271.009,A -85,B 0,C 180,E1 -10020.271,E2 -10020.271} C_VEL
LIN {X 0,Y 418.235,Z 271.012,A -85,B 0,C 180,E1 -10023.676,E2 -10023.676} C_VEL
LIN {X 0,Y 418.232,Z 271.015,A -85,B 0,C 180,E1 -10027.223,E2 -10027.223} C_VEL
LIN {X 0,Y 418.238,Z 271.011,A -85,B 0,C 180,E1 -10029.681,E2 -10029.681} C_VEL
LIN {X 0,Y 418.218,Z 271.011,A -85,B 0,C 180,E1 -10032.321,E2 -10032.321} C_VEL
LIN {X 0,Y 418.228,Z 271.015,A -85,B 0,C 180,E1 -10035.109,E2 -10035.109} C_VEL
LIN {X 0,Y 418.228,Z 271.011,A -85,B 0,C 180,E1 -10037.767,E2 -10037.767} C_VEL
LIN {X 0,Y 418.237,Z 271.009,A -85,B 0,C 180,E1 -10040.619,E2 -10040.619} C_VEL
LIN {X 0,Y 418.229,Z 271.01,A -85,B 0,C 180,E1 -10043.976,E2 -10043.976} C_VEL
LIN {X 0,Y 418.243,Z 271.014,A -85,B 0,C 180,E1 -10047.156,E2 -10047.156} C_VEL
LIN {X 0,Y 418.254,Z 271.01,A -85,B 0,C 180,E1 -10050.895,E2 -10050.895} C_VEL
LIN {X 0,Y 418.255,Z 271.006,A -85,B 0,C 180,E1 -10054.096,E2 -10054.096} C_VEL
LIN {X 0,Y 418.217,Z 271.017,A -85,B 0,C 180,E1 -10057.264,E2 -10057.264} C_VEL
LIN {X 0,Y 418.269,Z 271.005,A -85,B 0,C 180,E1 -10060.364,E2 -10060.364} C_VEL
LIN {X 0,Y 418.303,Z 271.004,A -85,B 0,C 180,E1 -10063.405,E2 -10063.405} C_VEL
LIN {X 0,Y 418.332,Z 271.003,A -85,B 0,C 180,E1 -10067,E2 -10067} C_VEL
LIN {X 0,Y 418.327,Z 270.998,A -85,B 0,C 180,E1 -10070.329,E2 -10070.329} C_VEL
LIN {X 0,Y 418.473,Z 270.984,A -85,B 0,C 180,E1 -10073.249,E2 -10073.249} C_VEL
LIN {X 0,Y 418.323,Z 271.003,A -85,B 0,C 180,E1 -10075.182,E2 -10075.182} C_VEL
LIN {X 0,Y 418.532,Z 270.972,A -85,B 0,C 180,E1 -10078.076,E2 -10078.076} C_VEL
LIN {X 0,Y 418.659,Z 270.956,A -85,B 0,C 180,E1 -10080.001,E2 -10080.001} C_VEL
LIN {X 0,Y 418.487,Z 270.983,A -85,B 0,C 180,E1 -10082.889,E2 -10082.889} C_VEL
LIN {X 0,Y 418.478,Z 270.983,A -85,B 0,C 180,E1 -10086.752,E2 -10086.752} C_VEL
LIN {X 0,Y 418.388,Z 270.994,A -85,B 0,C 180,E1 -10088.696,E2 -10088.696} C_VEL
LIN {X 0,Y 418.304,Z 271.001,A -85,B 0,C 180,E1 -10091.632,E2 -10091.632} C_VEL
LIN {X 0,Y 418.291,Z 271.005,A -85,B 0,C 180,E1 -10094.598,E2 -10094.598} C_VEL
LIN {X 0,Y 418.276,Z 271.004,A -85,B 0,C 180,E1 -10097.605,E2 -10097.605} C_VEL
LIN {X 0,Y 418.239,Z 271.013,A -85,B 0,C 180,E1 -10100.664,E2 -10100.664} C_VEL
LIN {X 0,Y 418.265,Z 271.005,A -85,B 0,C 180,E1 -10103.783,E2 -10103.783} C_VEL
LIN {X 0,Y 418.3,Z 271.005,A -85,B 0,C 180,E1 -10107.072,E2 -10107.072} C_VEL
LIN {X 0,Y 418.235,Z 271.01,A -85,B 0,C 180,E1 -10110.273,E2 -10110.273} C_VEL
LIN {X 0,Y 418.239,Z 271.008,A -85,B 0,C 180,E1 -10113.679,E2 -10113.679} C_VEL
LIN {X 0,Y 418.231,Z 271.012,A -85,B 0,C 180,E1 -10117.226,E2 -10117.226} C_VEL
LIN {X 0,Y 418.236,Z 271.008,A -85,B 0,C 180,E1 -10119.684,E2 -10119.684} C_VEL
LIN {X 0,Y 418.222,Z 271.013,A -85,B 0,C 180,E1 -10122.323,E2 -10122.323} C_VEL
LIN {X 0,Y 418.228,Z 271.013,A -85,B 0,C 180,E1 -10125.11,E2 -10125.11} C_VEL
LIN {X 0,Y 418.233,Z 271.009,A -85,B 0,C 180,E1 -10127.768,E2 -10127.768} C_VEL
LIN {X 0,Y 418.249,Z 271.014,A -85,B 0,C 180,E1 -10130.621,E2 -10130.621} C_VEL
LIN {X 0,Y 418.236,Z 271.01,A -85,B 0,C 180,E1 -10133.977,E2 -10133.977} C_VEL
